# B&R Automation Studio project TD52 (part 30)

```iecst
	(* W9254 Engine cooling water hydraulic pre-heating failure *)
	xMsg9254.Enable	   :=	(xEngType.Type3 OR xEngType.Type4 OR xEngType.Type6)
					AND		Para.bT_HW_Su_PreH_ECW_Active
					AND	(	(Para.iECW_PreH_Int_Visible = 5)					(* el.+hydr. pre-heating available *)
						 OR (	(Para.iECW_PreH_Int_Visible = 3)				(* only hydr. pre-heating available *)
							 AND NOT (Para.rT_ECW_HydrPreH_LimLo = 0.0)	)	);	(* monitoring deactivated if hydr. pre-heating only and Para.rT_ECW_HydrPreH_LimLo = 0.0 *)
	xMsg9254.Set 	   := 	IN_AG.tPB2MM.bParaSetupOk
					AND		bECW_HydrPreH_Dem
					AND (	((IN_AG.tT_ECW.Ai < rT_ECW_HydrPreH_LimLo) AND xSR_PreH_HeatUpDone.Q1)
						 OR	((IN_AG.tT_HW_Su_PreH_ECW.Ai < MM2VIS.rT_HW_Su_PreH_ECW_LimLo) AND IN_AG.tT_HW_Su_PreH_ECW.GoodQual)
						 OR	((IN_AG.tT_HW_Su_PreH_ECW.Ai > MM2VIS.rT_HW_Su_PreH_ECW_LimHi) AND IN_AG.tT_HW_Su_PreH_ECW.GoodQual)	);
	xMsg9254.PT	       := T#0s;
	xMsg9254.Prio 	   := 4;
	xMsg9254.RiskClass := 4;
	xMsg9254.Reset 	   := FALSE;
	xMsg9254();
	MM2VIS.bMsg9254    := xMsg9254.Q;

	(* W9255 Failure high temperature circuit pump 2 (redundant heating water pump) *)
	xMsg9255.Enable	   := Para.bRedHWP_Active;
	xMsg9255.Set 	   := bRedHWP_Fail AND ((iRedHWP_Fail = 2) OR (iRedHWP_Fail = 3));
	xMsg9255.PT	       := T#0s;
	xMsg9255.Prio 	   := 4;
	xMsg9255.RiskClass := 4;
	xMsg9255.Reset	   := FALSE;
	xMsg9255();
	MM2VIS.bMsg9255    := xMsg9255.Q;

	(* W9256 Failure low temperature circuit pump 3 (redundant charge cooler pump) *)
	xMsg9256.Enable	   := Para.bRedCCWP_Active;
	xMsg9256.Set 	   := bRedCCWP_Fail AND ((iRedCCWP_Fail = 2) OR (iRedCCWP_Fail = 3));
	xMsg9256.PT	       := T#0s;
	xMsg9256.Prio 	   := 4;
	xMsg9256.RiskClass := 4;
	xMsg9256.Reset	   := FALSE;
	xMsg9256();
	MM2VIS.bMsg9256    := xMsg9256.Q;

	(* W9257 Failure low temperature circuit pump 4 (redundant charge cooler 2 pump) *)
	xMsg9257.Enable	   := Para.bRedCC2WP_Active;
	xMsg9257.Set 	   := bRedCC2WP_Fail AND ((iRedCC2WP_Fail = 2) OR (iRedCC2WP_Fail = 3));
	xMsg9257.PT	       := T#0s;
	xMsg9257.Prio 	   := 4;
	xMsg9257.RiskClass := 4;
	xMsg9257.Reset	   := FALSE;
	xMsg9257();
	MM2VIS.bMsg9257    := xMsg9257.Q;

	(* W9258 Failure emergency cooling circuit pump 2 (redundant emergency cooler pump) *)
	xMsg9258.Enable	   := Para.bRedEmCWP_Active;
	xMsg9258.Set 	   := bRedEmCWP_Fail AND ((iRedEmCWP_Fail = 2) OR (iRedEmCWP_Fail = 3));
	xMsg9258.PT	       := T#0s;
	xMsg9258.Prio 	   := 4;
	xMsg9258.RiskClass := 4;
	xMsg9258.Reset	   := FALSE;
	xMsg9258();
	MM2VIS.bMsg9258    := xMsg9258.Q;

	(* W9279 Failure emergency cooling circuit pump 1 (emergency cooler pump) *)
	xTOF_EmCWP_Fail(IN:= IN_AG.tEmCWP_Op.Di OR bNoMon4BlackStart, PT:= T#10s);			(*pump operation feedback has to disappear for 10s to trigger warning, ignore feedback in case of black start*)
	xTON_EmCWP_Dem(IN:= IN_AG.bEmCWP_Dem, PT:= T#175s);
	HBT_8 := xTOF_EmCWP_Fail.Q OR (IN_AG.bEng_Aux_Dem AND IN_AG.bEmCWP_Dem AND HBT_8);	(*case 1: HBT_8 -> monitoring activated as soon as pump operation feedback is active for the first time*)

	xMsg9279.Enable	   := TRUE;
	IF NOT Para.bRedEmCWP_Active THEN
		xMsg9279.Set   := (xTON_EmCWP_Dem.Q OR HBT_8) AND NOT xTOF_EmCWP_Fail.Q AND IN_AG.bEmCWP_Dem;		(*case 2: xTON_EmCWP_Dem -> monitoring activated with delay after pump demand*)
	ELSE
		xMsg9279.Set   := bRedEmCWP_Fail AND ((iRedEmCWP_Fail = 1) OR (iRedEmCWP_Fail = 3));
	END_IF;
	xMsg9279.PT	       := T#2s;
	xMsg9279.Prio 	   := 4;
	xMsg9279.RiskClass := 4;
	xMsg9279.Reset	   := FALSE;
	xMsg9279();
	MM2VIS.bMsg9279    := xMsg9279.Q;

	(* W9280 Maximum number of failed post coolings for turbocharger exceeded; inspection of turbocharger required *)
	xMsg9280.Enable	   := FALSE AND IN_AG.tPB2MM.bParaSetupOk;
	xMsg9280.Set 	   := iCnt_TC_rel_A >= Para.iCnt_TC_Inspection_Hi;			(* if only one TC, counter for bank A is used *)
	xMsg9280.PT	       := T#0s;
	xMsg9280.Prio 	   := 4;
	xMsg9280.RiskClass := 4;
	xMsg9280.Reset	   := FALSE;
	xMsg9280();
	MM2VIS.bMsg9280    := xMsg9280.Q;

	(* W9281 Maximum number of failed post coolings for turbocharger at bank A exceeded; inspection of turbocharger required *)
	xMsg9281.Enable	   := xEngType.Type9 AND IN_AG.tPB2MM.bParaSetupOk;
	xMsg9281.Set 	   := iCnt_TC_rel_A >= Para.iCnt_TC_Inspection_Hi;
	xMsg9281.PT	       := T#0s;
	xMsg9281.Prio 	   := 4;
	xMsg9281.RiskClass := 4;
	xMsg9281.Reset	   := FALSE;
	xMsg9281();
	MM2VIS.bMsg9281    := xMsg9281.Q;

	(* W9282 Maximum number of failed post coolings for turbocharger at bank B exceeded; inspection of turbocharger required *)
	xMsg9282.Enable	   := xEngType.Type9 AND IN_AG.tPB2MM.bParaSetupOk;
	xMsg9282.Set 	   := iCnt_TC_rel_B >= Para.iCnt_TC_Inspection_Hi;
	xMsg9282.PT	       := T#0s;
	xMsg9282.Prio 	   := 4;
	xMsg9282.RiskClass := 4;
	xMsg9282.Reset	   := FALSE;
	xMsg9282();
	MM2VIS.bMsg9282    := xMsg9282.Q;

	(* W9283 Failed post cooling for turbocharger detected *)
	xMsg9283.Enable	   := NOT xEngType.Type2 AND IN_AG.tPB2MM.bParaSetupOk;
	xMsg9283.Set 	   := (EDGEPOS(IN_AG.tPB2MM.bSys_Run) AND iSt_TC_PwrInterrupt.0) OR EDGENEG(bTC_CoolDownInterrupt);
	xMsg9283.PT	       := T#0s;
	xMsg9283.Prio 	   := 4;
	xMsg9283.RiskClass := 4;
	xMsg9283.Reset	   := FALSE;
	xMsg9283();
	MM2VIS.bMsg9283    := xMsg9283.Q;

	(* W9303 Measuring signal failure air starter engagement pressure *)
	xMsg9303.Enable	   := xEngType.Type9;
	xMsg9303.Set 	   := bAMM_Pr_AirST_Engage_Ms;
	xMsg9303.PT	       := T#0s;
	xMsg9303.Prio 	   := 4;
	xMsg9303.RiskClass := 4;
	xMsg9303.Reset	   := FALSE;
	xMsg9303();
	MM2VIS.bMsg9303    := xMsg9303.Q;

	(* W9314 Engine cooling water pump circuit breaker tripped *)
	xMsg9314.Enable	   := IN_AG.tPB2MM.bParaSetupOk;
	xMsg9314.Set 	   := NOT IN_AG.tECWP_CB_On.Di;
	xMsg9314.PT	       := T#1s;
	xMsg9314.Prio 	   := 4;
	xMsg9314.RiskClass := 4;
	xMsg9314.Reset	   := FALSE;
	xMsg9314();
	MM2VIS.bMsg9314    := xMsg9314.Q;

	(* W9316 Measuring signal failure cooling water pressure after ECW pump 1 *)
	xMsg9316.Enable	   := Para.bDPr_ECWP_Mon_Active AND IN_AG.tPr_ECWaP1.Exist;
	xMsg9316.Set 	   := NOT IN_AG.tPr_ECWaP1.GoodQual;
	xMsg9316.PT	       := T#1s;
	xMsg9316.Prio 	   := 4;
	xMsg9316.RiskClass := 4;
	xMsg9316.Reset	   := FALSE;
	xMsg9316();
	MM2VIS.bMsg9316    := xMsg9316.Q;

	(* W9317 Measuring signal failure cooling water pressure after ECW pump 2 *)
	xMsg9317.Enable	   := Para.bDPr_ECWP_Mon_Active AND IN_AG.tPr_ECWaP2.Exist;
	xMsg9317.Set 	   := NOT IN_AG.tPr_ECWaP2.GoodQual;
	xMsg9317.PT	       := T#1s;
	xMsg9317.Prio 	   := 4;
	xMsg9317.RiskClass := 4;
	xMsg9317.Reset	   := FALSE;
	xMsg9317();
	MM2VIS.bMsg9317    := xMsg9317.Q;

	(* W9322 Fresh oil tank level low (2nd level switch) *)
	xMsg9322.Enable	   := IN_AG.tL_FreshOilTank_LoLo.GoodQual;
	xMsg9322.Set 	   := NOT IN_AG.tL_FreshOilTank_LoLo.Di;
	xMsg9322.PT	       := T#0s;
	xMsg9322.Prio 	   := 4;
	xMsg9322.RiskClass := 4;
	xMsg9322.Reset	   := FALSE;
	xMsg9322();
	MM2VIS.bMsg9322    := xMsg9322.Q;

	(* W9323 Fresh oil day tank level low *)
	xMsg9323.Enable	   := IN_AG.tPB2MM.bParaSetupOk;
	xMsg9323.Set 	   := (IN_AG.tL_DayOilTank_Lo.GoodQual AND NOT IN_AG.tL_DayOilTank_Lo.Di)
					   OR (IN_AG.tL_DayOilTank.GoodQual AND (MM2VIS.rV_DayOilTank < Para.rV_DayOilTank_LimLo) AND (Para.rV_DayOilTank_LimLo > 0)) ;		(*New at V4.12*)
	xMsg9323.PT	       := T#0s;
	xMsg9323.Prio 	   := 4;
	xMsg9323.RiskClass := 4;
	xMsg9323.Reset	   := FALSE;
	xMsg9323();
	MM2VIS.bMsg9323    := xMsg9323.Q;

	(* W9324 Fresh oil day tank level low (2nd level switch) *)
	xMsg9324.Enable	   := IN_AG.tL_DayOilTank_LoLo.GoodQual;
	xMsg9324.Set 	   := NOT IN_AG.tL_DayOilTank_LoLo.Di;
	xMsg9324.PT	       := T#0s;
	xMsg9324.Prio 	   := 4;
	xMsg9324.RiskClass := 4;
	xMsg9324.Reset	   := FALSE;
	xMsg9324();
	MM2VIS.bMsg9324    := xMsg9324.Q;

	(* W9325 Overfill prevention device fresh oil day tank tripped *)
	xMsg9325.Enable	   := IN_AG.tOF_DayOilTank.GoodQual;
	xMsg9325.Set 	   := NOT IN_AG.tOF_DayOilTank.Di;
	xMsg9325.PT	       := T#0s;
	xMsg9325.Prio 	   := 4;
	xMsg9325.RiskClass := 4;
	xMsg9325.Reset	   := FALSE;
	xMsg9325();
	MM2VIS.bMsg9325    := xMsg9325.Q;

	(* W9326 Waste oil day tank level high *)
	xMsg9326.Enable	   := IN_AG.tL_WasteOilDayTank_Hi.GoodQual;
	xMsg9326.Set 	   := NOT IN_AG.tL_WasteOilDayTank_Hi.Di;
	xMsg9326.PT	       := T#0s;
	xMsg9326.Prio 	   := 4;
	xMsg9326.RiskClass := 4;
	xMsg9326.Reset	   := FALSE;
	xMsg9326();
	MM2VIS.bMsg9326    := xMsg9326.Q;

	(* W9327 Overfill prevention device waste oil day tank tripped *)
	xMsg9327.Enable	   := IN_AG.tOF_WasteOilDayTank.GoodQual;
	xMsg9327.Set 	   := NOT IN_AG.tOF_WasteOilDayTank.Di;
	xMsg9327.PT	       := T#0s;
	xMsg9327.Prio 	   := 4;
	xMsg9327.RiskClass := 4;
	xMsg9327.Reset	   := FALSE;
	xMsg9327();
	MM2VIS.bMsg9327    := xMsg9327.Q;

	(* W9328 Fresh oil pump oil pressure maximum *)
	xMsg9328.Enable	   := IN_AG.tPS_FreshOilPump_Hi.GoodQual;
	xMsg9328.Set 	   := NOT IN_AG.tPS_FreshOilPump_Hi.Di;
	xMsg9328.PT	       := T#0s;
	xMsg9328.Prio 	   := 4;
	xMsg9328.RiskClass := 4;
	xMsg9328.Reset	   := FALSE;
	xMsg9328();
	MM2VIS.bMsg9328    := xMsg9328.Q;

	(* W9332 Take oil sample *)
	xMsg9332.Enable	   := Para.bEO_Management_Active AND IN_AG.tPB2MM.bParaSetupOk;
	xMsg9332.Set 	   := bMsg9332_set;
	xMsg9332.PT	       := T#0s;
	xMsg9332.Prio 	   := 4;
	xMsg9332.RiskClass := 4;
	xMsg9332.Reset	   := TRUE;
	xMsg9332();
	MM2VIS.bMsg9332    := xMsg9332.Q;

	(* W9333 Take coolant sample *)
	xMsg9333.Enable	   := Para.bCW_Management_Active AND IN_AG.tPB2MM.bParaSetupOk;
	xMsg9333.Set 	   := bMsg9333_set;
	xMsg9333.PT	       := T#0s;
	xMsg9333.Prio 	   := 4;
	xMsg9333.RiskClass := 4;
	xMsg9333.Reset	   := TRUE;
	xMsg9333();
	MM2VIS.bMsg9333    := xMsg9333.Q;

	(* W9334 Buffer battery 1 voltage low *)
	xMsg9334.Enable	   := IN_AG.tPB2MM.bParaSetupOk AND ((Para.iBatMon_Mode = 1) OR (Para.iBatMon_Mode = 2));
	xMsg9334.Set 	   := bAMM_U_BufferBat1_Lo;
	xMsg9334.PT	       := T#0s;
	xMsg9334.Prio 	   := 4;
	xMsg9334.RiskClass := 4;
	xMsg9334.Reset	   := FALSE;
	xMsg9334();
	MM2VIS.bMsg9334    := xMsg9334.Q;

	(* W9335 Buffer battery 2 voltage low *)
	xMsg9335.Enable	   := IN_AG.tPB2MM.bParaSetupOk AND (Para.iBatMon_Mode = 2);
	xMsg9335.Set 	   := bAMM_U_BufferBat2_Lo;
	xMsg9335.PT	       := T#0s;
	xMsg9335.Prio 	   := 4;
	xMsg9335.RiskClass := 4;
	xMsg9335.Reset	   := FALSE;
	xMsg9335();
	MM2VIS.bMsg9335    := xMsg9335.Q;

	(* W9336 Battery charging device malfunction *)
	xMsg9336.Enable	   := IN_AG.tPB2MM.bParaSetupOk;
	xMsg9336.Set 	   := NOT IN_AG.tBatChargeDev_Ok.Di;
	xMsg9336.PT	       := T#10s;
	xMsg9336.Prio 	   := 4;
	xMsg9336.RiskClass := 4;
	xMsg9336.Reset	   := FALSE;
	xMsg9336();
	MM2VIS.bMsg9336    := xMsg9336.Q;

	(* W9352 Oil quality sensor - Measurement signal failure, return to regular sampling interval *)
	xMsg9352.Enable	   := (Para.iOQS_Config = 1) AND IN_AG.tPB2MM.bParaSetupOk AND NOT IN_AG.bSimWinMOD_Active;
	xMsg9352.Set 	   := bAMM_OQS_OC_MSF;
	xMsg9352.PT	       := T#0s;
	xMsg9352.Prio 	   := 4;
	xMsg9352.RiskClass := 4;
	xMsg9352.Reset	   := FALSE;
	xMsg9352();
	MM2VIS.bMsg9352    := xMsg9352.Q;

	(* W9353 Oil quality sensor - Oil quality warning, return to regular sampling interval *)
	xMsg9353.Enable	   := (Para.iOQS_Config = 1) AND IN_AG.tPB2MM.bParaSetupOk AND NOT IN_AG.bSimWinMOD_Active;
	xMsg9353.Set 	   := bAMM_OQS_OC_ValueLo;
	xMsg9353.PT	       := T#0s;
	xMsg9353.Prio 	   := 4;
	xMsg9353.RiskClass := 4;
	xMsg9353.Reset	   := FALSE;
	xMsg9353();
	MM2VIS.bMsg9353    := xMsg9353.Q;

	(* W9354 Oil quality sensor  Critical oil quality warning, return to regular sampling interval *)
	xMsg9354.Enable	   := (Para.iOQS_Config = 1) AND IN_AG.tPB2MM.bParaSetupOk AND NOT IN_AG.bSimWinMOD_Active;
	xMsg9354.Set 	   := bAMM_OQS_OC_ValueLo1;
	xMsg9354.PT	       := T#0s;
	xMsg9354.Prio 	   := 4;
	xMsg9354.RiskClass := 4;
	xMsg9354.Reset	   := FALSE;
	xMsg9354();
	MM2VIS.bMsg9354    := xMsg9354.Q;

	(* W9355 Oil quality sensor  Increased oil aging, return to regular sampling interval *)
	xMsg9355.Enable	   := (Para.iOQS_Config = 1) AND IN_AG.tPB2MM.bParaSetupOk AND NOT IN_AG.bSimWinMOD_Active;
	xMsg9355.Set 	   := bAMM_OQS_OC_TendencyHi;
	xMsg9355.PT	       := T#0s;
	xMsg9355.Prio 	   := 4;
	xMsg9355.RiskClass := 4;
	xMsg9355.Reset	   := FALSE;
	xMsg9355();
	MM2VIS.bMsg9355    := xMsg9355.Q;

	(* W9356 Oil quality sensor - Critical oil aging, return to regular sampling interval *)
	xMsg9356.Enable	   := (Para.iOQS_Config = 1) AND IN_AG.tPB2MM.bParaSetupOk AND NOT IN_AG.bSimWinMOD_Active;
	xMsg9356.Set 	   := bAMM_OQS_OC_TendencyHi1;
	xMsg9356.PT	       := T#0s;
	xMsg9356.Prio 	   := 4;
	xMsg9356.RiskClass := 4;
	xMsg9356.Reset	   := FALSE;
	xMsg9356();
	MM2VIS.bMsg9356    := xMsg9356.Q;

	(* W9357 Control battery voltage low *)
	xMsg9357.Enable	   := IN_AG.tPB2MM.bParaSetupOk AND (iNr_CtrlBat_Used > 0);
	xMsg9357.Set 	   := bAMM_U_CtrlBat_Lo_Coll;
	xMsg9357.PT	       := T#0s;
	xMsg9357.Prio 	   := 4;
	xMsg9357.RiskClass := 4;
	xMsg9357.Reset	   := FALSE;
	xMsg9357();
	MM2VIS.bMsg9357    := xMsg9357.Q;

	(* W9358 Control battery charging device malfunction *)
	bAMM_CtrlBat_ChargeDev_Fail		:=	FALSE;
	FOR iIdx_CtrlBat := 1 TO iNum_CtrlBatMon DO
		bAMM_CtrlBat_ChargeDev_Fail	:=	NOT IN_AG.tCtrlBat_ChargeDev_Ok[iIdx_CtrlBat].Di OR bAMM_CtrlBat_ChargeDev_Fail;
		IF NOT IN_AG.tCtrlBat_ChargeDev_Ok[iIdx_CtrlBat].Di THEN
			MM2VIS.sCtrlBat_ChargeDev_LocFault	:=	IN_AG.sLocIdent_CtrlBatMon[iIdx_CtrlBat];
		END_IF;
	END_FOR;
	xMsg9358.Enable	   := IN_AG.tPB2MM.bParaSetupOk AND (iNr_CtrlBat_Used > 0);
	xMsg9358.Set 	   := bAMM_CtrlBat_ChargeDev_Fail;
	xMsg9358.PT	       := T#10s;
	xMsg9358.Prio 	   := 4;
	xMsg9358.RiskClass := 4;
	xMsg9358.Reset	   := FALSE;
	xMsg9358();
	MM2VIS.bMsg9358    := xMsg9358.Q;

	(* W9359 Oil pressure before centrifuge (oil filter unit) minimum *)
	xMsg9359.Enable	   := Para.bOilFiltUnit_Exist AND Para.bPr_OFUbCentrifuge_Active;
	xMsg9359.Set 	   := bAMM_Pr_OFUbCentrifuge_Lo;
	xMsg9359.PT	       := T#2s;
	xMsg9359.Prio 	   := 4;
	xMsg9359.RiskClass := 4;
	xMsg9359.Reset	   := FALSE;
	xMsg9359();
	MM2VIS.bMsg9359    := xMsg9359.Q;

	(*W9362 Fresh Oil Tank Signal Failure V4.12 *)
	xMsg9362.Enable		:=  Para.bOilTankMonitoring AND Para.rFreshOilTank_Type > 0;
	xMsg9362.Set 	   := NOT IN_AG.tL_FreshOilTank.GoodQual;
	xMsg9362.PT	       := T#2s;
	xMsg9362.Prio 	   := 4;
	xMsg9362.RiskClass := 4;
	xMsg9362.Reset	   := FALSE;
	xMsg9362();
	MM2VIS.bMsg9362    := xMsg9362.Q;

	(*W9363 Waste Oil Tank Signal Failure V4.12 *)
	xMsg9363.Enable		:=  Para.bOilTankMonitoring AND Para.rWasteOilTank_Type > 0;
	xMsg9363.Set 	   := NOT IN_AG.tL_WasteOilTank.GoodQual;
	xMsg9363.PT	       := T#2s;
	xMsg9363.Prio 	   := 4;
	xMsg9363.RiskClass := 4;
	xMsg9363.Reset	   := FALSE;
	xMsg9363();
	MM2VIS.bMsg9363    := xMsg9363.Q;

	(*W9364 Fresh Oil Tank Signal Failure V4.12 *)
	xMsg9364.Enable		:=  Para.bOilTankMonitoring AND Para.rDayOilTank_Type > 0;
	xMsg9364.Set 	   := NOT IN_AG.tL_DayOilTank.GoodQual;
	xMsg9364.PT	       := T#2s;
	xMsg9364.Prio 	   := 4;
	xMsg9364.RiskClass := 4;
	xMsg9364.Reset	   := FALSE;
	xMsg9364();
	MM2VIS.bMsg9364    := xMsg9364.Q;

	(*W9369 Failure auxiliaries supply voltage engine V4.12 *)
	xMsg9369.Enable		:= IN_AG.tPB2MM.bParaSetupOk;
	xMsg9369.Set		:= (NOT IN_AG.tAuxV_Eng_ok.Di) AND IN_AG.tAuxV_Eng_ok.GoodQual AND IN_AG.tMnsOk.Di AND IN_AG.tMnsOk.GoodQual;
	xMsg9369.PT			:= T#1m;
	xMsg9369.Prio		:= 4;
	xMsg9369.RiskClass	:= 4;
	xMsg9369.Reset		:= FALSE;
	xMsg9369();
	MM2VIS.bMsg9369    := xMsg9369.Q;

	(*W9378 Oil refill volume maximum *)
	xMsg9378.Enable		:= IN_AG.tPB2MM.bParaSetupOk;
	xMsg9378.Set		:= bAMM_Vol_OilRefill_Hi;
	xMsg9378.PT			:= T#0s;
	xMsg9378.Prio		:= 4;
	xMsg9378.RiskClass	:= 4;
	xMsg9378.Reset		:= FALSE;
	xMsg9378();
	MM2VIS.bMsg9378    	:= xMsg9378.Q;

	(*W9390 Oil temperature before engine start too low *)
	xMsg9390.Enable		:= IN_AG.tPB2MM.bParaSetupOk;
	xMsg9390.Set		:= bAMM_T_EO_PreH_EngStart_Lo;
	xMsg9390.PT			:= T#0s;
	xMsg9390.Prio		:= 4;
	xMsg9390.RiskClass	:= 4;
	xMsg9390.Reset		:= NOT bAMM_T_EO_PreH_EngStart_Lo;
	xMsg9390();
	MM2VIS.bMsg9390    	:= xMsg9390.Q;

	(* A9435 Fire detection system - System failure *)
	xMsg9435.Enable	   	:= IN_AG.tPB2MM.bParaSetupOk AND IN_AG.bSafetyPLC_Active;			(* SAFETY PLC *)
	xMsg9435.Set	  	:= NOT IN_AG.tFireSysErr.Di;
	xMsg9435.PT	       	:= T#240s;
	xMsg9435.Prio	   	:= 3;
	xMsg9435.RiskClass	:= 4;
	xMsg9435.Reset	   	:= FALSE;
	xMsg9435();
	MM2VIS.bMsg9435		:= xMsg9435.Q;

	(* A9436 Gas detection system - System failure *)
	xMsg9436.Enable	   	:= IN_AG.tPB2MM.bParaSetupOk AND IN_AG.bSafetyPLC_Active;			(* SAFETY PLC *)
	xMsg9436.Set	  	:= NOT IN_AG.tGasSysErr.Di;
	xMsg9436.PT	       	:= T#240s;
	xMsg9436.Prio	   	:= 3;
	xMsg9436.RiskClass	:= 4;
	xMsg9436.Reset	   	:= FALSE;
	xMsg9436();
	MM2VIS.bMsg9436		:= xMsg9436.Q;

	(* W9560 Fire detection system - System failure *)
	xMsg9560.Enable	   	:= IN_AG.tPB2MM.bParaSetupOk AND IN_AG.bSafetyPLC_Active;			(* SAFETY PLC *)
	xMsg9560.Set	  	:= NOT IN_AG.tFireSysErr.Di;
	xMsg9560.PT	       	:= T#0s;
	xMsg9560.Prio	   	:= 4;
	xMsg9560.RiskClass	:= 4;
	xMsg9560.Reset	   	:= FALSE;
	xMsg9560();
	MM2VIS.bMsg9560		:= xMsg9560.Q;

	(* W9561 Gas detection system - System failure *)
	xMsg9561.Enable	   	:= IN_AG.tPB2MM.bParaSetupOk AND IN_AG.bSafetyPLC_Active;			(* SAFETY PLC *)
	xMsg9561.Set	  	:= NOT IN_AG.tGasSysErr.Di;
	xMsg9561.PT	       	:= T#0s;
	xMsg9561.Prio	   	:= 4;
	xMsg9561.RiskClass	:= 4;
	xMsg9561.Reset	   	:= FALSE;
	xMsg9561();
	MM2VIS.bMsg9561		:= xMsg9561.Q;

	(*---------------------------------------------------------------------------*)
	(* operating messages > AMM *)

	(* B1249 starter engine on *)
	xMsg1249.Enable		:=	TRUE;
	xMsg1249.Set		:= 	(OUT_AG.bEng_Start AND xEngType.Type9) OR (OUT_AG.tEleStarter_Dem.Do AND NOT xEngType.Type9);
	xMsg1249.Reset		:=	TRUE;
	xMsg1249();
	MM2VIS.bMsg1249		:=	xMsg1249.Q;

	(* B1250 starter engine off *)
	xMsg1250.Enable		:=	IN_AG.tPB2MM.bSys_Run;
	xMsg1250.Set		:=	NOT MM2VIS.bMsg1249;
	xMsg1250.Reset		:=	TRUE;
	xMsg1250();
	MM2VIS.bMsg1250		:= xMsg1250.Q;

	(* B1257 demand engine cooling water pump on *)
	xMsg1257.Enable		:=	TRUE;
	xMsg1257.Set		:=	    OUT_AG.tECWP1Dem.Do;
	xMsg1257.Reset		:=	TRUE;
	xMsg1257();
	MM2VIS.bMsg1257		:= xMsg1257.Q;

	(* B1258 demand engine cooling water pump off *)
	xMsg1258.Enable		:=	IN_AG.tPB2MM.bSys_Run;
	xMsg1258.Set		:=	NOT OUT_AG.tECWP1Dem.Do;
	xMsg1258.Reset		:=	TRUE;
	xMsg1258();
	MM2VIS.bMsg1258		:= xMsg1258.Q;

	(* B1259 demand oil pump on *)
	xMsg1259.Enable		:=	TRUE;
	xMsg1259.Set		:=	OUT_AG.tEOP1AC_Dem.Do;
	xMsg1259.Reset		:=	TRUE;
	xMsg1259();
	MM2VIS.bMsg1259		:= xMsg1259.Q;

	(* B1260 demand oil pump off *)
	xMsg1260.Enable		:=	IN_AG.tPB2MM.bSys_Run;
	xMsg1260.Set		:=	NOT OUT_AG.tEOP1AC_Dem.Do;
	xMsg1260.Reset		:=	TRUE;
	xMsg1260();
	MM2VIS.bMsg1260		:= xMsg1260.Q;

	(* B1261 demand oil pump (DC) on *)
	xMsg1261.Enable		:=	NOT xEngType.Type9;
	xMsg1261.Set		:=	    OUT_AG.tEOP1DC_Dem.Do;
	xMsg1261.Reset		:=	TRUE;
	xMsg1261();
	MM2VIS.bMsg1261		:= xMsg1261.Q;

	(* B1262 demand oil pump (DC) off *)
	xMsg1262.Enable		:=	IN_AG.tPB2MM.bSys_Run AND NOT xEngType.Type9;
	xMsg1262.Set		:=	NOT OUT_AG.tEOP1DC_Dem.Do;
	xMsg1262.Reset		:=	TRUE;
	xMsg1262();
	MM2VIS.bMsg1262		:= xMsg1262.Q;

	(* B1263 demand turbo charger oil pump on *)
	xMsg1263.Enable		:=	TRUE;
	xMsg1263.Set		:=  OUT_AG.tTC_EOP_On.Do OR OUT_AG.tTC_EOP_OnUSV.Do;
	xMsg1263.Reset		:=	TRUE;
	xMsg1263();
	MM2VIS.bMsg1263		:= xMsg1263.Q;

	(* B1264 demand turbo charger oil pump off *)
	xMsg1264.Enable		:=	IN_AG.tPB2MM.bSys_Run AND xEngType.Type9;
	xMsg1264.Set		:=	NOT OUT_AG.tTC_EOP_On.Do AND NOT OUT_AG.tTC_EOP_OnUSV.Do;
	xMsg1264.Reset		:=	TRUE;
	xMsg1264();
	MM2VIS.bMsg1264		:= xMsg1264.Q;

	(* B1281 demand engine cooling water preheating pump on *)
	xMsg1281.Enable		:=	TRUE;
	xMsg1281.Set		:=	    OUT_AG.tECWP_PreH_Dem.Do;
	xMsg1281.Reset		:=	TRUE;
	xMsg1281();
	MM2VIS.bMsg1281		:= xMsg1281.Q;

	(* B1282 demand engine cooling water preheating pump off *)
	xMsg1282.Enable		:=	IN_AG.tPB2MM.bSys_Run;
	xMsg1282.Set		:=	NOT OUT_AG.tECWP_PreH_Dem.Do;
	xMsg1282.Reset		:=	TRUE;
	xMsg1282();
	MM2VIS.bMsg1282		:= xMsg1282.Q;

	(* B1292 Manual operating auxiliaries control (Handbedienebene) active *)
	xMsg1292.Enable		:=	IN_AG.tPB2MM.bSys_Run;
	xMsg1292.Set		:=	bMsg1292_Set;
	xMsg1292.Reset		:=	TRUE;
	xMsg1292();
	MM2VIS.bMsg1292		:= xMsg1292.Q;

	(* B2809 preheating valve opened *)
	xMsg2809.Enable		:=	IN_AG.tPB2MM.bSys_Run;
	xMsg2809.Set		:=	IN_AG.tECW_PreHV_Opened.Di;
	xMsg2809.Reset		:=	TRUE;
	xMsg2809();
	MM2VIS.bMsg2809		:= xMsg2809.Q;

	(* B2810 Preheating valve closed *)
	xMsg2810.Enable		:=	bECW_PreHV_Active;
	xMsg2810.Set		:=	IN_AG.tECW_PreHV_Closed.Di;
	xMsg2810.Reset		:=	TRUE;
	xMsg2810();
	MM2VIS.bMsg2810		:= xMsg2810.Q;

	(* B2931 Active Cooling Program in operation *)
	xMsg2931.Enable		:=	Para.bACP_Enable;
	xMsg2931.Set		:=	bACP_Start AND NOT bACP_Cmp;
	xMsg2931.Reset		:=	TRUE;
	xMsg2931();
	MM2VIS.bMsg2931		:= xMsg2931.Q;

	(* B2932 Active Cooling Program finished *)
	xMsg2932.Enable		:=	Para.bACP_Enable;
	xMsg2932.Set		:=	bACP_Cmp;
	xMsg2932.Reset		:=	TRUE;
	xMsg2932();
	MM2VIS.bMsg2932		:= xMsg2932.Q;

	(* B2933 Active Cooling Program cancelled *)
	xF_TRIG_ACP_Start(CLK := bACP_Start);
	xMsg2933.Enable		:=	Para.bACP_Enable;
	xMsg2933.Set		:=	xF_TRIG_ACP_Start.Q AND NOT bACP_Cmp;
	xMsg2933.Reset		:=	TRUE;
	xMsg2933();
	MM2VIS.bMsg2933		:= xMsg2933.Q;

	(* B2956 Demand engine oil preheating valve open *)
	xMsg2956.Enable		:=	IN_AG.tPB2MM.bSys_Run
						AND xEngType.Type9;
	xMsg2956.Set		:=	OUT_AG.tEOF_PreheatRel.Do;
	xMsg2956.Reset		:=	TRUE;
	xMsg2956();
	MM2VIS.bMsg2956		:= xMsg2956.Q;

	(* B2957 Demand engine oil preheating valve close *)
	xMsg2957.Enable		:=	IN_AG.tPB2MM.bSys_Run
						AND xEngType.Type9;
	xMsg2957.Set		:=	NOT OUT_AG.tEOF_PreheatRel.Do;
	xMsg2957.Reset		:=	TRUE;
	xMsg2957();
	MM2VIS.bMsg2957		:= xMsg2957.Q;

	(* B2978 Blow-by blower on *)
	xMsg2978.Enable		:=	xEngType.Type9;
	xMsg2978.Set		:=	OUT_AG.tBbBlower.Do;
	xMsg2978.Reset		:=	TRUE;
	xMsg2978();
	MM2VIS.bMsg2978		:= xMsg2978.Q;

	(* B2979 Blow-by blower off *)
	xMsg2979.Enable		:=	xEngType.Type9;
	xMsg2979.Set		:=	NOT OUT_AG.tBbBlower.Do;
	xMsg2979.Reset		:=	TRUE;
	xMsg2979();
	MM2VIS.bMsg2979		:= xMsg2979.Q;

	(* B3300 blocking acknowledgement by starter temperature *)
	xMsg3300.Enable		:=	TRUE;
	xMsg3300.Set		:=	OUT_AG.bLockAckStarter;
	xMsg3300.Reset		:=	TRUE;
	xMsg3300();
	MM2VIS.bMsg3300		:= xMsg3300.Q;

	(* B9001 Oil sample taken *)
	xMsg9001.Enable		:=	Para.bEO_Management_Active AND IN_AG.tPB2MM.bParaSetupOk;
	xMsg9001.Set		:=	bMsg9001_set;
	xMsg9001.Reset		:=	TRUE;
	xMsg9001();
	MM2VIS.bMsg9001		:= xMsg9001.Q;

	(* B9002 Oil exchanged *)
	xMsg9002.Enable		:=	Para.bEO_Management_Active AND IN_AG.tPB2MM.bParaSetupOk;
	xMsg9002.Set		:=	bMsg9002_set;
	xMsg9002.Reset		:=	TRUE;
	xMsg9002();
	MM2VIS.bMsg9002		:= xMsg9002.Q;

	(* B9003 Coolant sample taken *)
	xMsg9003.Enable		:=	Para.bCW_Management_Active AND IN_AG.tPB2MM.bParaSetupOk;
	xMsg9003.Set		:=	bMsg9003_set;
	xMsg9003.Reset		:=	TRUE;
	xMsg9003();
	MM2VIS.bMsg9003		:= xMsg9003.Q;

	(* B9048 Coolant exchanged *)
	xMsg9048.Enable		:=	Para.bCW_Management_Active AND IN_AG.tPB2MM.bParaSetupOk;
	xMsg9048.Set		:=	bMsg9048_set;
	xMsg9048.Reset		:=	TRUE;
	xMsg9048();
	MM2VIS.bMsg9048		:= xMsg9048.Q;

	(* B9067 Oil sampling interval extended *)
	xMsg9067.Enable		:=	(Para.iOQS_Config = 1) AND IN_AG.tPB2MM.bParaSetupOk AND NOT IN_AG.bSimWinMOD_Active;
	xMsg9067.Set		:=	bOpMsg_ExtendOilSampleOh;
	xMsg9067.Reset		:=	TRUE;
	xMsg9067();
	MM2VIS.bMsg9067		:= xMsg9067.Q;

	(* B9069 Buffer battery test in progress *)
	xMsg9069.Enable		:= IN_AG.tPB2MM.bParaSetupOk AND (Para.iBatMon_Mode > 0);
	xMsg9069.Set		:= MM2VIS.bBatMon_TestRunning;
	xMsg9069.Reset		:= TRUE;
	xMsg9069();
	MM2VIS.bMsg9069		:= xMsg9069.Q;

	(* B9070 Control battery test in progress *)
	xMsg9070.Enable		:= IN_AG.tPB2MM.bParaSetupOk AND (iNr_CtrlBat_Used > 0);
	xMsg9070.Set		:= MM2VIS.bCtrlBatMon_TestRunning;
	xMsg9070.Reset		:= TRUE;
	xMsg9070();
	MM2VIS.bMsg9070		:= xMsg9070.Q;

	(* B9074 Tooth to tooth position *)
	xMsg9074.Enable		:= IN_AG.tPB2MM.bParaSetupOk;
	xMsg9074.Set		:= FALSE; // warning message for tooth to tooth detection. Not used yet, already set up in the HMI
	xMsg9074.Reset		:= TRUE;
	xMsg9074();
	MM2VIS.bMsg9074		:= xMsg9074.Q;

	(* B9088 Purge cranking cycle successful *)
	xMsg9088.Enable		:= IN_AG.tPB2MM.bParaSetupOk;
	xMsg9088.Set		:= (bStartScavSflMsg AND xEngType.Type3) OR (bMsg9088_T6_set AND xEngType.Type6);
	xMsg9088.Reset		:= TRUE;
	xMsg9088();
	MM2VIS.bMsg9088 	:= xMsg9088.Q;

	(* B9089 Starter motor 1 did not engage *)
	xMsg9089.Enable		:= IN_AG.tPB2MM.bParaSetupOk AND Para.rU_StarterMon_LimLo <> 0.0;
	xMsg9089.Set		:= bEleStarterFail_Num[1];
	xMsg9089.Reset		:= TRUE;
	xMsg9089();
	MM2VIS.bMsg9089		:= xMsg9089.Q;

	(* B9090 Starter motor 2 did not engage *)
	xMsg9090.Enable		:= IN_AG.tPB2MM.bParaSetupOk AND Para.rU_StarterMon_LimLo <> 0.0;
	xMsg9090.Set		:= bEleStarterFail_Num[2];
	xMsg9090.Reset		:= TRUE;
	xMsg9090();
	MM2VIS.bMsg9090		:= xMsg9090.Q;

	(* B9091 Starter motor 3 did not engage *)
	xMsg9091.Enable		:= IN_AG.tPB2MM.bParaSetupOk AND Para.rU_StarterMon_LimLo <> 0.0;
	xMsg9091.Set		:= bEleStarterFail_Num[3];
	xMsg9091.Reset		:= TRUE;
	xMsg9091();
	MM2VIS.bMsg9091		:= xMsg9091.Q;

	(* B9096 Starter overheated *)
	xMsg9096.Enable		:= IN_AG.tPB2MM.bParaSetupOk AND xEngType.Type6;
	xMsg9096.Set		:= bMsg9096_set AND bMsg9096_enable;
	xMsg9096.Reset		:= TRUE;
	xMsg9096();
	MM2VIS.bMsg9096		:= xMsg9096.Q;
	MM2VIS.iNum_Msg9096	:= bMsg9096_iTi_ST_UntRelDur;

	(* B9097 Purge cranking cycle initiated *)
	xMsg9097.Enable		:= IN_AG.tPB2MM.bParaSetupOk AND xEngType.Type6;
	xMsg9097.Set		:= bMsg9097_set;
	xMsg9097.Reset		:= TRUE;
	xMsg9097();
	MM2VIS.bMsg9097		:= xMsg9097.Q;

	(*W9513 Failure engine oil refilling *)
	xMsg9513.Enable 	:= IN_AG.tPB2MM.bParaSetupOk ;
	xMsg9513.Set 		:= bAMM_9513;
	xMsg9513.PT 		:= Para.tiEO_Refill_TimeMax;
	xMsg9513.Prio 		:= 4;
	xMsg9513.Reset 		:= FALSE;
	xMsg9513();
	MM2VIS.bMsg9513 	:= xMsg9513.Q;

	(* B template
	xMsg.Enable		:=	TRUE;
	xMsg.Set		:=	bBool;
	xMsg.Reset		:=	TRUE;
	xMsg();
	MM2VIS.bMsg		:=	xMsg.Q;
	*)

	(*---------------------------------------------------------------------------*)
	(* general alarms for further module operations *)
	bGnlTrip1		:= OUT_AG.tAG2AB.bGnlTrip1   OR IN_AG.tAB2AG.bGnlTrip1;
	bGnlTrip2		:= OUT_AG.tAG2AB.bGnlTrip2   OR IN_AG.tAB2AG.bGnlTrip2;
	bGnlTrip3		:= OUT_AG.tAG2AB.bGnlTrip3   OR IN_AG.tAB2AG.bGnlTrip3;
	bGnlWarning		:= OUT_AG.tAG2AB.bGnlWarning OR IN_AG.tAB2AG.bGnlWarning;

	bGnlTrip		:= bGnlTrip1 OR bGnlTrip2 OR bGnlTrip3;

	(*******************************************************************************)

END_PROGRAM
```

#### MsgAGInit.st
```iecst
(*******************************************************************************
Msg_AG	 			 alarms generation auxiliaries general

This code is confidential and proprietary to the INNIO Company.
It may not be used in any form, or reproduced in any manner,
without written permission of the INNIO Company.
Copyright, INNIO Company, 2022

Customized modifications: -
------------------------

History:
-------
V0.00.0	29.07.2011	lettenb.	new
V4.12.0	21.12.2022	Perktold	added W9369 Failure auxiliaries supply voltage engine

Instructions for use:
--------------------
1) declare alarm with function block "Msg"

2) use template to create a new alarm, substitue 0000 by message number:

	xMsg0000.Num		:=	0000;					alarm number
	xMsg0000.AmmSysAdr	:=  iAdrAmmBase2MM;			do not change
	xMsg0000.AmmOutAdr	:=  iAdrMM2AmmBase;			do not change

3) 	set alarm number

Outstandings:
------------
(*******************************************************************************)
PROGRAM _INIT

	bPLC_Startup := FALSE;

	iAdrAmmBase2MM		:=  ADR(IN_AG.tAB2AG);
	iAdrMM2AmmBase		:=  ADR(OUT_AG.tAG2AB);

	(*---------------------------------------------------------------------------*)
	xMsg1017.Num		:=	1017;
	xMsg1017.AmmInAdr	:=  iAdrAmmBase2MM;
	xMsg1017.AmmOutAdr	:=  iAdrMM2AmmBase;

	xMsg1018.Num		:=  1018;
	xMsg1018.AmmInAdr	:=  iAdrAmmBase2MM;
	xMsg1018.AmmOutAdr	:=  iAdrMM2AmmBase;

	xMsg1020.Num		:=  1020;
	xMsg1020.AmmInAdr	:=  iAdrAmmBase2MM;
	xMsg1020.AmmOutAdr	:=  iAdrMM2AmmBase;

	xMsg1023.Num		:=  1023;
	xMsg1023.AmmInAdr	:=  iAdrAmmBase2MM;
	xMsg1023.AmmOutAdr	:=  iAdrMM2AmmBase;

	xMsg1043.Num		:=	1043;
	xMsg1043.AmmInAdr	:=  iAdrAmmBase2MM;
	xMsg1043.AmmOutAdr	:=  iAdrMM2AmmBase;

	xMsg1051.Num		:=	1051;
	xMsg1051.AmmInAdr	:=  iAdrAmmBase2MM;
	xMsg1051.AmmOutAdr	:=  iAdrMM2AmmBase;

	xMsg1052.Num		:=  1052;
	xMsg1052.AmmInAdr	:=  iAdrAmmBase2MM;
	xMsg1052.AmmOutAdr	:=  iAdrMM2AmmBase;

	xMsg1053.Num		:=  1053;
	xMsg1053.AmmInAdr	:=  iAdrAmmBase2MM;
	xMsg1053.AmmOutAdr	:=  iAdrMM2AmmBase;

	xMsg1054.Num		:=  1054;
	xMsg1054.AmmInAdr	:=  iAdrAmmBase2MM;
	xMsg1054.AmmOutAdr	:=  iAdrMM2AmmBase;

	xMsg1059.Num		:=	1059;
	xMsg1059.AmmInAdr	:=  iAdrAmmBase2MM;
	xMsg1059.AmmOutAdr	:=  iAdrMM2AmmBase;

	xMsg1060.Num		:=  1060;
	xMsg1060.AmmInAdr	:=  iAdrAmmBase2MM;
	xMsg1060.AmmOutAdr	:=  iAdrMM2AmmBase;

	xMsg1090.Num		:=  1090;
	xMsg1090.AmmInAdr	:=  iAdrAmmBase2MM;
	xMsg1090.AmmOutAdr	:=  iAdrMM2AmmBase;

	xMsg1091.Num		:=  1091;
	xMsg1091.AmmInAdr	:=  iAdrAmmBase2MM;
	xMsg1091.AmmOutAdr	:=  iAdrMM2AmmBase;

	xMsg1100.Num		:=  1100;
	xMsg1100.AmmInAdr	:=  iAdrAmmBase2MM;
	xMsg1100.AmmOutAdr	:=  iAdrMM2AmmBase;

	xMsg1101.Num		:=  1101;
	xMsg1101.AmmInAdr	:=  iAdrAmmBase2MM;
	xMsg1101.AmmOutAdr	:=  iAdrMM2AmmBase;

	xMsg1120.Num		:=  1120;
	xMsg1120.AmmInAdr	:=  iAdrAmmBase2MM;
	xMsg1120.AmmOutAdr	:=  iAdrMM2AmmBase;

	xMsg1129.Num		:=  1129;
	xMsg1129.AmmInAdr	:=  iAdrAmmBase2MM;
	xMsg1129.AmmOutAdr	:=  iAdrMM2AmmBase;

	xMsg1137.Num		:=  1137;
	xMsg1137.AmmInAdr	:=  iAdrAmmBase2MM;
	xMsg1137.AmmOutAdr	:=  iAdrMM2AmmBase;

	xMsg1139.Num		:=  1139;
	xMsg1139.AmmInAdr	:=  iAdrAmmBase2MM;
	xMsg1139.AmmOutAdr	:=  iAdrMM2AmmBase;

	xMsg1140.Num		:=  1140;
	xMsg1140.AmmInAdr	:=  iAdrAmmBase2MM;
	xMsg1140.AmmOutAdr	:=  iAdrMM2AmmBase;

	xMsg1148.Num		:=  1148;
	xMsg1148.AmmInAdr	:=  iAdrAmmBase2MM;
	xMsg1148.AmmOutAdr	:=  iAdrMM2AmmBase;

	xMsg1159.Num		:=  1159;
	xMsg1159.AmmInAdr	:=  iAdrAmmBase2MM;
	xMsg1159.AmmOutAdr	:=  iAdrMM2AmmBase;

	xMsg1160.Num		:=  1160;
	xMsg1160.AmmInAdr	:=  iAdrAmmBase2MM;
	xMsg1160.AmmOutAdr	:=  iAdrMM2AmmBase;

	xMsg1166.Num		:=	1166;
	xMsg1166.AmmInAdr	:=  iAdrAmmBase2MM;
	xMsg1166.AmmOutAdr	:=  iAdrMM2AmmBase;

	xMsg1249.Num		:=	1249;
	xMsg1249.AmmInAdr	:=  iAdrAmmBase2MM;
	xMsg1249.AmmOutAdr	:=  iAdrMM2AmmBase;

	xMsg1250.Num		:=	1250;
	xMsg1250.AmmInAdr	:=  iAdrAmmBase2MM;
	xMsg1250.AmmOutAdr	:=  iAdrMM2AmmBase;

	xMsg1257.Num		:=	1257;
	xMsg1257.AmmInAdr	:=  iAdrAmmBase2MM;
	xMsg1257.AmmOutAdr	:=  iAdrMM2AmmBase;

	xMsg1258.Num		:=	1258;
	xMsg1258.AmmInAdr	:=  iAdrAmmBase2MM;
	xMsg1258.AmmOutAdr	:=  iAdrMM2AmmBase;

	xMsg1259.Num		:=	1259;
	xMsg1259.AmmInAdr	:=  iAdrAmmBase2MM;
	xMsg1259.AmmOutAdr	:=  iAdrMM2AmmBase;

	xMsg1260.Num		:=	1260;
	xMsg1260.AmmInAdr	:=  iAdrAmmBase2MM;
	xMsg1260.AmmOutAdr	:=  iAdrMM2AmmBase;

	xMsg1261.Num		:=	1261;
	xMsg1261.AmmInAdr	:=  iAdrAmmBase2MM;
	xMsg1261.AmmOutAdr	:=  iAdrMM2AmmBase;

	xMsg1262.Num		:=	1262;
	xMsg1262.AmmInAdr	:=  iAdrAmmBase2MM;
	xMsg1262.AmmOutAdr	:=  iAdrMM2AmmBase;

	xMsg1263.Num		:=	1263;
	xMsg1263.AmmInAdr	:=  iAdrAmmBase2MM;
	xMsg1263.AmmOutAdr	:=  iAdrMM2AmmBase;

	xMsg1264.Num		:=	1264;
	xMsg1264.AmmInAdr	:=  iAdrAmmBase2MM;
	xMsg1264.AmmOutAdr	:=  iAdrMM2AmmBase;

	xMsg1281.Num		:=	1281;
	xMsg1281.AmmInAdr	:=  iAdrAmmBase2MM;
	xMsg1281.AmmOutAdr	:=  iAdrMM2AmmBase;

	xMsg1282.Num		:=	1282;
	xMsg1282.AmmInAdr	:=  iAdrAmmBase2MM;
	xMsg1282.AmmOutAdr	:=  iAdrMM2AmmBase;

	xMsg1292.Num		:=	1292;
	xMsg1292.AmmInAdr	:=  iAdrAmmBase2MM;
	xMsg1292.AmmOutAdr	:=  iAdrMM2AmmBase;

	xMsg2102.Num		:=	2102;
	xMsg2102.AmmInAdr	:=  iAdrAmmBase2MM;
	xMsg2102.AmmOutAdr	:=  iAdrMM2AmmBase;

	xMsg2103.Num		:=	2103;
	xMsg2103.AmmInAdr	:=  iAdrAmmBase2MM;
	xMsg2103.AmmOutAdr	:=  iAdrMM2AmmBase;

	xMsg2114.Num		:=  2114;
	xMsg2114.AmmInAdr	:=  iAdrAmmBase2MM;
	xMsg2114.AmmOutAdr	:=  iAdrMM2AmmBase;

	xMsg2118.Num		:=  2118;
	xMsg2118.AmmInAdr	:=  iAdrAmmBase2MM;
	xMsg2118.AmmOutAdr	:=  iAdrMM2AmmBase;

	xMsg2201.Num		:=  2201;
	xMsg2201.AmmInAdr	:=  iAdrAmmBase2MM;
	xMsg2201.AmmOutAdr	:=  iAdrMM2AmmBase;

	xMsg2213.Num		:=	2213;
	xMsg2213.AmmInAdr	:=  iAdrAmmBase2MM;
	xMsg2213.AmmOutAdr	:=  iAdrMM2AmmBase;

	xMsg2224.Num		:=	2224;
	xMsg2224.AmmInAdr	:=  iAdrAmmBase2MM;
	xMsg2224.AmmOutAdr	:=  iAdrMM2AmmBase;

	xMsg2233.Num		:=	2233;
	xMsg2233.AmmInAdr	:=  iAdrAmmBase2MM;
	xMsg2233.AmmOutAdr	:=  iAdrMM2AmmBase;

	xMsg2234.Num		:=	2234;
	xMsg2234.AmmInAdr	:=  iAdrAmmBase2MM;
	xMsg2234.AmmOutAdr	:=  iAdrMM2AmmBase;

	xMsg2238.Num		:=	2238;
	xMsg2238.AmmInAdr	:=  iAdrAmmBase2MM;
	xMsg2238.AmmOutAdr	:=  iAdrMM2AmmBase;

	xMsg2242.Num		:=	2242;
	xMsg2242.AmmInAdr	:=  iAdrAmmBase2MM;
	xMsg2242.AmmOutAdr	:=  iAdrMM2AmmBase;

	xMsg2260.Num		:=	2260;
	xMsg2260.AmmInAdr	:=  iAdrAmmBase2MM;
	xMsg2260.AmmOutAdr	:=  iAdrMM2AmmBase;

	xMsg2263.Num		:=  2263;
	xMsg2263.AmmInAdr	:=  iAdrAmmBase2MM;
	xMsg2263.AmmOutAdr	:=  iAdrMM2AmmBase;

	xMsg2264.Num		:=  2264;
	xMsg2264.AmmInAdr	:=  iAdrAmmBase2MM;
	xMsg2264.AmmOutAdr	:=  iAdrMM2AmmBase;

	xMsg2265.Num		:=  2265;
	xMsg2265.AmmInAdr	:=  iAdrAmmBase2MM;
	xMsg2265.AmmOutAdr	:=  iAdrMM2AmmBase;

	xMsg2266.Num		:=  2266;
	xMsg2266.AmmInAdr	:=  iAdrAmmBase2MM;
	xMsg2266.AmmOutAdr	:=  iAdrMM2AmmBase;

	xMsg2267.Num		:=  2267;
	xMsg2267.AmmInAdr	:=  iAdrAmmBase2MM;
	xMsg2267.AmmOutAdr	:=  iAdrMM2AmmBase;

	xMsg2268.Num		:=  2268;
	xMsg2268.AmmInAdr	:=  iAdrAmmBase2MM;
	xMsg2268.AmmOutAdr	:=  iAdrMM2AmmBase;

	xMsg2269.Num		:=  2269;
	xMsg2269.AmmInAdr	:=  iAdrAmmBase2MM;
	xMsg2269.AmmOutAdr	:=  iAdrMM2AmmBase;

	xMsg2284.Num		:=	2284;
	xMsg2284.AmmInAdr	:=  iAdrAmmBase2MM;
	xMsg2284.AmmOutAdr	:=  iAdrMM2AmmBase;

	xMsg2291.Num		:=  2291;
	xMsg2291.AmmInAdr	:=  iAdrAmmBase2MM;
	xMsg2291.AmmOutAdr	:=  iAdrMM2AmmBase;

	xMsg2292.Num		:=  2292;
	xMsg2292.AmmInAdr	:=  iAdrAmmBase2MM;
	xMsg2292.AmmOutAdr	:=  iAdrMM2AmmBase;

	xMsg2304.Num		:=	2304;
	xMsg2304.AmmInAdr	:=  iAdrAmmBase2MM;
	xMsg2304.AmmOutAdr	:=  iAdrMM2AmmBase;

	xMsg2332.Num		:=	2332;
	xMsg2332.AmmInAdr	:=  iAdrAmmBase2MM;
	xMsg2332.AmmOutAdr	:=  iAdrMM2AmmBase;

	xMsg2333.Num		:=	2333;
	xMsg2333.AmmInAdr	:=  iAdrAmmBase2MM;
	xMsg2333.AmmOutAdr	:=  iAdrMM2AmmBase;

	xMsg2348.Num		:=	2348;
	xMsg2348.AmmInAdr	:=  iAdrAmmBase2MM;
	xMsg2348.AmmOutAdr	:=  iAdrMM2AmmBase;

	xMsg2349.Num		:=	2349;
	xMsg2349.AmmInAdr	:=  iAdrAmmBase2MM;
	xMsg2349.AmmOutAdr	:=  iAdrMM2AmmBase;

	xMsg2350.Num		:=	2350;
	xMsg2350.AmmInAdr	:=  iAdrAmmBase2MM;
	xMsg2350.AmmOutAdr	:=  iAdrMM2AmmBase;

	xMsg2351.Num		:=	2351;
	xMsg2351.AmmInAdr	:=  iAdrAmmBase2MM;
	xMsg2351.AmmOutAdr	:=  iAdrMM2AmmBase;

	xMsg2352.Num		:=	2352;
	xMsg2352.AmmInAdr	:=  iAdrAmmBase2MM;
	xMsg2352.AmmOutAdr	:=  iAdrMM2AmmBase;

	xMsg2353.Num		:=	2353;
	xMsg2353.AmmInAdr	:=  iAdrAmmBase2MM;
	xMsg2353.AmmOutAdr	:=  iAdrMM2AmmBase;

	xMsg2355.Num		:=	2355;
	xMsg2355.AmmInAdr	:=  iAdrAmmBase2MM;
	xMsg2355.AmmOutAdr	:=  iAdrMM2AmmBase;

	xMsg2359.Num		:=	2359;
	xMsg2359.AmmInAdr	:=  iAdrAmmBase2MM;
	xMsg2359.AmmOutAdr	:=  iAdrMM2AmmBase;

	xMsg2360.Num		:=	2360;
	xMsg2360.AmmInAdr	:=  iAdrAmmBase2MM;
	xMsg2360.AmmOutAdr	:=  iAdrMM2AmmBase;

	xMsg2361.Num		:=	2361;
	xMsg2361.AmmInAdr	:=  iAdrAmmBase2MM;
	xMsg2361.AmmOutAdr	:=  iAdrMM2AmmBase;

	xMsg2376.Num		:=	2376;
	xMsg2376.AmmInAdr	:=  iAdrAmmBase2MM;
	xMsg2376.AmmOutAdr	:=  iAdrMM2AmmBase;

	xMsg2377.Num		:=	2377;
	xMsg2377.AmmInAdr	:=  iAdrAmmBase2MM;
	xMsg2377.AmmOutAdr	:=  iAdrMM2AmmBase;

	xMsg2378.Num		:=	2378;
	xMsg2378.AmmInAdr	:=  iAdrAmmBase2MM;
	xMsg2378.AmmOutAdr	:=  iAdrMM2AmmBase;

	xMsg2379.Num		:=	2379;
	xMsg2379.AmmInAdr	:=  iAdrAmmBase2MM;
	xMsg2379.AmmOutAdr	:=  iAdrMM2AmmBase;

	xMsg2382.Num		:=	2382;
	xMsg2382.AmmInAdr	:=  iAdrAmmBase2MM;
	xMsg2382.AmmOutAdr	:=  iAdrMM2AmmBase;

	xMsg2421.Num		:=	2421;
	xMsg2421.AmmInAdr	:=  iAdrAmmBase2MM;
	xMsg2421.AmmOutAdr	:=  iAdrMM2AmmBase;

	xMsg2422.Num		:=  2422;
	xMsg2422.AmmInAdr	:=  iAdrAmmBase2MM;
	xMsg2422.AmmOutAdr	:=  iAdrMM2AmmBase;

	xMsg2423.Num		:=	2423;//SWAT920/1
	xMsg2423.AmmInAdr	:=  iAdrAmmBase2MM;
	xMsg2423.AmmOutAdr	:=  iAdrMM2AmmBase;

	xMsg2424.Num		:=	2424;//SWAT920/2.2
	xMsg2424.AmmInAdr	:=  iAdrAmmBase2MM;
	xMsg2424.AmmOutAdr	:=  iAdrMM2AmmBase;

	xMsg2425.Num		:=	2425;//SWAT920/2.2
	xMsg2425.AmmInAdr	:=  iAdrAmmBase2MM;
	xMsg2425.AmmOutAdr	:=  iAdrMM2AmmBase;

	xMsg2426.Num		:=	2426;//SWAT920/2.2
	xMsg2426.AmmInAdr	:=  iAdrAmmBase2MM;
	xMsg2426.AmmOutAdr	:=  iAdrMM2AmmBase;

	xMsg2427.Num		:=	2427;
	xMsg2427.AmmInAdr	:=  iAdrAmmBase2MM;
	xMsg2427.AmmOutAdr	:=  iAdrMM2AmmBase;

	xMsg2431.Num		:=	2431;//SWAT920/1
	xMsg2431.AmmInAdr	:=  iAdrAmmBase2MM;
	xMsg2431.AmmOutAdr	:=  iAdrMM2AmmBase;

	xMsg2432.Num		:=	2432;//SWAT920/1
	xMsg2432.AmmInAdr	:=  iAdrAmmBase2MM;
	xMsg2432.AmmOutAdr	:=  iAdrMM2AmmBase;

	xMsg2433.Num		:=	2433;//SWAT920/1
	xMsg2433.AmmInAdr	:=  iAdrAmmBase2MM;
	xMsg2433.AmmOutAdr	:=  iAdrMM2AmmBase;

	xMsg2434.Num		:=	2434;
	xMsg2434.AmmInAdr	:=  iAdrAmmBase2MM;
	xMsg2434.AmmOutAdr	:=  iAdrMM2AmmBase;

	xMsg2435.Num		:=	2435;//SWAT920/2
	xMsg2435.AmmInAdr	:=  iAdrAmmBase2MM;
	xMsg2435.AmmOutAdr	:=  iAdrMM2AmmBase;

	xMsg2459.Num		:=  2459;
	xMsg2459.AmmInAdr	:=  iAdrAmmBase2MM;
	xMsg2459.AmmOutAdr	:=  iAdrMM2AmmBase;

	xMsg2473.Num		:=  2473;
	xMsg2473.AmmInAdr	:=  iAdrAmmBase2MM;
	xMsg2473.AmmOutAdr	:=  iAdrMM2AmmBase;

	xMsg2475.Num		:=  2475;
	xMsg2475.AmmInAdr	:=  iAdrAmmBase2MM;
	xMsg2475.AmmOutAdr	:=  iAdrMM2AmmBase;

	xMsg2524.Num		:=	2524;
	xMsg2524.AmmInAdr	:=  iAdrAmmBase2MM;
	xMsg2524.AmmOutAdr	:=  iAdrMM2AmmBase;

	xMsg2534.Num		:=	2534;
	xMsg2534.AmmInAdr	:=  iAdrAmmBase2MM;
	xMsg2534.AmmOutAdr	:=  iAdrMM2AmmBase;

	xMsg2545.Num		:=  2545;
	xMsg2545.AmmInAdr	:=  iAdrAmmBase2MM;
	xMsg2545.AmmOutAdr	:=  iAdrMM2AmmBase;

	xMsg2554.Num		:=	2554;
	xMsg2554.AmmInAdr	:=  iAdrAmmBase2MM;
	xMsg2554.AmmOutAdr	:=  iAdrMM2AmmBase;

	xMsg2557.Num		:=	2557;//SWAT920/2.2
	xMsg2557.AmmInAdr	:=  iAdrAmmBase2MM;
	xMsg2557.AmmOutAdr	:=  iAdrMM2AmmBase;

	xMsg2558.Num		:=  2558;
	xMsg2558.AmmInAdr	:=  iAdrAmmBase2MM;
	xMsg2558.AmmOutAdr	:=  iAdrMM2AmmBase;

	xMsg2559.Num 		:=  2559;
	xMsg2559.AmmInAdr 	:=  iAdrAmmBase2MM;
	xMsg2559.AmmOutAdr 	:=  iAdrMM2AmmBase;

	xMsg2560.Num		:=  2560;
	xMsg2560.AmmInAdr	:=  iAdrAmmBase2MM;
	xMsg2560.AmmOutAdr	:=  iAdrMM2AmmBase;

	xMsg2571.Num		:=  2571;
	xMsg2571.AmmInAdr	:=  iAdrAmmBase2MM;
	xMsg2571.AmmOutAdr	:=  iAdrMM2AmmBase;

	xMsg2572.Num		:=  2572;
	xMsg2572.AmmInAdr	:=  iAdrAmmBase2MM;
	xMsg2572.AmmOutAdr	:=  iAdrMM2AmmBase;

	xMsg2576.Num		:=	2576;
	xMsg2576.AmmInAdr	:=  iAdrAmmBase2MM;
	xMsg2576.AmmOutAdr	:=  iAdrMM2AmmBase;

	xMsg2579.Num		:=	2579;
	xMsg2579.AmmInAdr	:=  iAdrAmmBase2MM;
	xMsg2579.AmmOutAdr	:=  iAdrMM2AmmBase;

	xMsg2582.Num		:=	2582;
	xMsg2582.AmmInAdr	:=  iAdrAmmBase2MM;
	xMsg2582.AmmOutAdr	:=  iAdrMM2AmmBase;

	xMsg2587.Num		:=	2587;
	xMsg2587.AmmInAdr	:=  iAdrAmmBase2MM;
	xMsg2587.AmmOutAdr	:=  iAdrMM2AmmBase;

	xMsg2589.Num		:=  2589;
	xMsg2589.AmmInAdr	:=  iAdrAmmBase2MM;
	xMsg2589.AmmOutAdr	:=  iAdrMM2AmmBase;

	xMsg2590.Num		:=  2590;
	xMsg2590.AmmInAdr	:=  iAdrAmmBase2MM;
	xMsg2590.AmmOutAdr	:=  iAdrMM2AmmBase;

	xMsg2591.Num		:=  2591;
	xMsg2591.AmmInAdr	:=  iAdrAmmBase2MM;
	xMsg2591.AmmOutAdr	:=  iAdrMM2AmmBase;

	xMsg2592.Num		:=  2592;
	xMsg2592.AmmInAdr	:=  iAdrAmmBase2MM;
	xMsg2592.AmmOutAdr	:=  iAdrMM2AmmBase;

	xMsg2594.Num		:=  2594;
	xMsg2594.AmmInAdr	:=  iAdrAmmBase2MM;
	xMsg2594.AmmOutAdr	:=  iAdrMM2AmmBase;

	xMsg2595.Num		:=  2595;
	xMsg2595.AmmInAdr	:=  iAdrAmmBase2MM;
	xMsg2595.AmmOutAdr	:=  iAdrMM2AmmBase;

	xMsg2596.Num		:=  2596;
	xMsg2596.AmmInAdr	:=  iAdrAmmBase2MM;
	xMsg2596.AmmOutAdr	:=  iAdrMM2AmmBase;

	xMsg2597.Num		:=	2597;
	xMsg2597.AmmInAdr	:=  iAdrAmmBase2MM;
	xMsg2597.AmmOutAdr	:=  iAdrMM2AmmBase;

	xMsg2598.Num		:=	2598;
	xMsg2598.AmmInAdr	:=  iAdrAmmBase2MM;
	xMsg2598.AmmOutAdr	:=  iAdrMM2AmmBase;

	xMsg2599.Num		:=	2599;
	xMsg2599.AmmInAdr	:=  iAdrAmmBase2MM;
	xMsg2599.AmmOutAdr	:=  iAdrMM2AmmBase;

	xMsg2600.Num		:=	2600;
	xMsg2600.AmmInAdr	:=  iAdrAmmBase2MM;
	xMsg2600.AmmOutAdr	:=  iAdrMM2AmmBase;

	xMsg2602.Num		:=	2602;
	xMsg2602.AmmInAdr	:=  iAdrAmmBase2MM;
	xMsg2602.AmmOutAdr	:=  iAdrMM2AmmBase;

	xMsg2603.Num		:=	2603;
	xMsg2603.AmmInAdr	:=  iAdrAmmBase2MM;
	xMsg2603.AmmOutAdr	:=  iAdrMM2AmmBase;

	xMsg2604.Num		:=	2604;
	xMsg2604.AmmInAdr	:=  iAdrAmmBase2MM;
	xMsg2604.AmmOutAdr	:=  iAdrMM2AmmBase;

	xMsg2605.Num		:=	2605;
	xMsg2605.AmmInAdr	:=  iAdrAmmBase2MM;
	xMsg2605.AmmOutAdr	:=  iAdrMM2AmmBase;

	xMsg2606.Num		:=	2606;
	xMsg2606.AmmInAdr	:=  iAdrAmmBase2MM;
	xMsg2606.AmmOutAdr	:=  iAdrMM2AmmBase;

	xMsg2608.Num		:=	2608;
	xMsg2608.AmmInAdr	:=  iAdrAmmBase2MM;
	xMsg2608.AmmOutAdr	:=  iAdrMM2AmmBase;

	xMsg2613.Num		:=	2613;
	xMsg2613.AmmInAdr	:=  iAdrAmmBase2MM;
	xMsg2613.AmmOutAdr	:=  iAdrMM2AmmBase;

	xMsg2624.Num		:=	2624;
	xMsg2624.AmmInAdr	:=  iAdrAmmBase2MM;
	xMsg2624.AmmOutAdr	:=  iAdrMM2AmmBase;

	xMsg2625.Num		:=	2625;
	xMsg2625.AmmInAdr	:=  iAdrAmmBase2MM;
	xMsg2625.AmmOutAdr	:=  iAdrMM2AmmBase;

	xMsg2627.Num		:=	2627;
	xMsg2627.AmmInAdr	:=  iAdrAmmBase2MM;
	xMsg2627.AmmOutAdr	:=  iAdrMM2AmmBase;

	xMsg2628.Num		:=	2628;
	xMsg2628.AmmInAdr	:=  iAdrAmmBase2MM;
	xMsg2628.AmmOutAdr	:=  iAdrMM2AmmBase;

	xMsg2629.Num		:=	2629;
	xMsg2629.AmmInAdr	:=  iAdrAmmBase2MM;
	xMsg2629.AmmOutAdr	:=  iAdrMM2AmmBase;

	xMsg2636.Num		:=	2636;
	xMsg2636.AmmInAdr	:=  iAdrAmmBase2MM;
	xMsg2636.AmmOutAdr	:=  iAdrMM2AmmBase;

	xMsg2642.Num		:=	2642;
	xMsg2642.AmmInAdr	:=  iAdrAmmBase2MM;
	xMsg2642.AmmOutAdr	:=  iAdrMM2AmmBase;

	xMsg2643.Num		:=	2643;
	xMsg2643.AmmInAdr	:=  iAdrAmmBase2MM;
	xMsg2643.AmmOutAdr	:=  iAdrMM2AmmBase;

	xMsg2644.Num		:=	2644;
	xMsg2644.AmmInAdr	:=  iAdrAmmBase2MM;
	xMsg2644.AmmOutAdr	:=  iAdrMM2AmmBase;

	xMsg2645.Num		:=	2645;
	xMsg2645.AmmInAdr	:=  iAdrAmmBase2MM;
	xMsg2645.AmmOutAdr	:=  iAdrMM2AmmBase;

	xMsg2646.Num		:=	2646;
	xMsg2646.AmmInAdr	:=  iAdrAmmBase2MM;
	xMsg2646.AmmOutAdr	:=  iAdrMM2AmmBase;

	xMsg2648.Num		:=	2648;
	xMsg2648.AmmInAdr	:=  iAdrAmmBase2MM;
	xMsg2648.AmmOutAdr	:=  iAdrMM2AmmBase;

	xMsg2649.Num 		:= 	2649;
	xMsg2649.AmmInAdr 	:= iAdrAmmBase2MM;
	xMsg2649.AmmOutAdr 	:= iAdrMM2AmmBase;

	xMsg2650.Num 		:= 	2650;
	xMsg2650.AmmInAdr 	:= iAdrAmmBase2MM;
	xMsg2650.AmmOutAdr 	:= iAdrMM2AmmBase;

	xMsg2651.Num 		:= 	2651;
	xMsg2651.AmmInAdr 	:= iAdrAmmBase2MM;
	xMsg2651.AmmOutAdr 	:= iAdrMM2AmmBase;

	xMsg2652.Num 		:= 	2652;
	xMsg2652.AmmInAdr 	:= iAdrAmmBase2MM;
	xMsg2652.AmmOutAdr 	:= iAdrMM2AmmBase;

	xMsg2653.Num 		:= 	2653;
	xMsg2653.AmmInAdr 	:= iAdrAmmBase2MM;
	xMsg2653.AmmOutAdr 	:= iAdrMM2AmmBase;

	xMsg2654.Num 		:= 	2654;
	xMsg2654.AmmInAdr 	:= iAdrAmmBase2MM;
	xMsg2654.AmmOutAdr 	:= iAdrMM2AmmBase;

	xMsg2666.Num		:=	2666;
	xMsg2666.AmmInAdr	:=  iAdrAmmBase2MM;
	xMsg2666.AmmOutAdr	:=  iAdrMM2AmmBase;

	xMsg2689.Num		:=	2689;
	xMsg2689.AmmInAdr	:=  iAdrAmmBase2MM;
	xMsg2689.AmmOutAdr	:=  iAdrMM2AmmBase;

	xMsg2722.Num		:=	2722;
	xMsg2722.AmmInAdr	:=  iAdrAmmBase2MM;
	xMsg2722.AmmOutAdr	:=  iAdrMM2AmmBase;

	xMsg2723.Num		:=	2723;
	xMsg2723.AmmInAdr	:=  iAdrAmmBase2MM;
	xMsg2723.AmmOutAdr	:=  iAdrMM2AmmBase;

	xMsg2724.Num		:=	2724;
	xMsg2724.AmmInAdr	:=  iAdrAmmBase2MM;
	xMsg2724.AmmOutAdr	:=  iAdrMM2AmmBase;

	xMsg2725.Num		:=	2725;
	xMsg2725.AmmInAdr	:=  iAdrAmmBase2MM;
	xMsg2725.AmmOutAdr	:=  iAdrMM2AmmBase;

	xMsg2726.Num		:=	2726;
	xMsg2726.AmmInAdr	:=  iAdrAmmBase2MM;
	xMsg2726.AmmOutAdr	:=  iAdrMM2AmmBase;

	xMsg2727.Num		:=	2727;
	xMsg2727.AmmInAdr	:=  iAdrAmmBase2MM;
	xMsg2727.AmmOutAdr	:=  iAdrMM2AmmBase;

	xMsg2728.Num		:=	2728;
	xMsg2728.AmmInAdr	:=  iAdrAmmBase2MM;
	xMsg2728.AmmOutAdr	:=  iAdrMM2AmmBase;

	xMsg2729.Num		:=	2729;
	xMsg2729.AmmInAdr	:=  iAdrAmmBase2MM;
	xMsg2729.AmmOutAdr	:=  iAdrMM2AmmBase;

	xMsg2737.Num		:=	2737;
	xMsg2737.AmmInAdr	:=  iAdrAmmBase2MM;
	xMsg2737.AmmOutAdr	:=  iAdrMM2AmmBase;

	xMsg2738.Num		:=	2738;
	xMsg2738.AmmInAdr	:=  iAdrAmmBase2MM;
	xMsg2738.AmmOutAdr	:=  iAdrMM2AmmBase;

	xMsg2739.Num		:=	2739;
	xMsg2739.AmmInAdr	:=  iAdrAmmBase2MM;
	xMsg2739.AmmOutAdr	:=  iAdrMM2AmmBase;

	xMsg2740.Num		:=	2740;
	xMsg2740.AmmInAdr	:=  iAdrAmmBase2MM;
	xMsg2740.AmmOutAdr	:=  iAdrMM2AmmBase;

	xMsg2741.Num		:=	2741;
	xMsg2741.AmmInAdr	:=  iAdrAmmBase2MM;
	xMsg2741.AmmOutAdr	:=  iAdrMM2AmmBase;

	xMsg2742.Num		:=	2742;
	xMsg2742.AmmInAdr	:=  iAdrAmmBase2MM;
	xMsg2742.AmmOutAdr	:=  iAdrMM2AmmBase;

	xMsg2754.Num		:=	2754;
	xMsg2754.AmmInAdr	:=  iAdrAmmBase2MM;
	xMsg2754.AmmOutAdr	:=  iAdrMM2AmmBase;

	xMsg2755.Num		:=	2755;
	xMsg2755.AmmInAdr	:=  iAdrAmmBase2MM;
	xMsg2755.AmmOutAdr	:=  iAdrMM2AmmBase;

	xMsg2756.Num		:=	2756;
	xMsg2756.AmmInAdr	:=  iAdrAmmBase2MM;
	xMsg2756.AmmOutAdr	:=  iAdrMM2AmmBase;

	xMsg2757.Num		:=	2757;
	xMsg2757.AmmInAdr	:=  iAdrAmmBase2MM;
	xMsg2757.AmmOutAdr	:=  iAdrMM2AmmBase;

	xMsg2758.Num		:=	2758;
	xMsg2758.AmmInAdr	:=  iAdrAmmBase2MM;
	xMsg2758.AmmOutAdr	:=  iAdrMM2AmmBase;

	xMsg2759.Num		:=	2759;
	xMsg2759.AmmInAdr	:=  iAdrAmmBase2MM;
	xMsg2759.AmmOutAdr	:=  iAdrMM2AmmBase;

	xMsg2760.Num		:=	2760;
	xMsg2760.AmmInAdr	:=  iAdrAmmBase2MM;
	xMsg2760.AmmOutAdr	:=  iAdrMM2AmmBase;

	xMsg2761.Num		:=	2761;
	xMsg2761.AmmInAdr	:=  iAdrAmmBase2MM;
	xMsg2761.AmmOutAdr	:=  iAdrMM2AmmBase;

	xMsg2762.Num		:=	2762;
	xMsg2762.AmmInAdr	:=  iAdrAmmBase2MM;
	xMsg2762.AmmOutAdr	:=  iAdrMM2AmmBase;

	xMsg2770.Num		:=	2770;
	xMsg2770.AmmInAdr	:=  iAdrAmmBase2MM;
	xMsg2770.AmmOutAdr	:=  iAdrMM2AmmBase;

	xMsg2771.Num		:=	2771;
	xMsg2771.AmmInAdr	:=  iAdrAmmBase2MM;
	xMsg2771.AmmOutAdr	:=  iAdrMM2AmmBase;

	xMsg2772.Num		:=	2772;
	xMsg2772.AmmInAdr	:=  iAdrAmmBase2MM;
	xMsg2772.AmmOutAdr	:=  iAdrMM2AmmBase;

	xMsg2773.Num		:=	2773;
	xMsg2773.AmmInAdr	:=  iAdrAmmBase2MM;
	xMsg2773.AmmOutAdr	:=  iAdrMM2AmmBase;

	xMsg2774.Num		:=	2774;
	xMsg2774.AmmInAdr	:=  iAdrAmmBase2MM;
	xMsg2774.AmmOutAdr	:=  iAdrMM2AmmBase;

	xMsg2775.Num		:=	2775;
	xMsg2775.AmmInAdr	:=  iAdrAmmBase2MM;
	xMsg2775.AmmOutAdr	:=  iAdrMM2AmmBase;

	xMsg2776.Num		:=	2776;
	xMsg2776.AmmInAdr	:=  iAdrAmmBase2MM;
	xMsg2776.AmmOutAdr	:=  iAdrMM2AmmBase;

	xMsg2777.Num		:=	2777;
	xMsg2777.AmmInAdr	:=  iAdrAmmBase2MM;
	xMsg2777.AmmOutAdr	:=  iAdrMM2AmmBase;

	xMsg2778.Num		:=	2778;
	xMsg2778.AmmInAdr	:=  iAdrAmmBase2MM;
	xMsg2778.AmmOutAdr	:=  iAdrMM2AmmBase;

	xMsg2781.Num		:=	2781;
	xMsg2781.AmmInAdr	:=  iAdrAmmBase2MM;
	xMsg2781.AmmOutAdr	:=  iAdrMM2AmmBase;

	xMsg2782.Num		:=	2782;
	xMsg2782.AmmInAdr	:=  iAdrAmmBase2MM;
	xMsg2782.AmmOutAdr	:=  iAdrMM2AmmBase;

	xMsg2783.Num		:=	2783;
	xMsg2783.AmmInAdr	:=  iAdrAmmBase2MM;
	xMsg2783.AmmOutAdr	:=  iAdrMM2AmmBase;

	xMsg2784.Num		:=	2784;
	xMsg2784.AmmInAdr	:=  iAdrAmmBase2MM;
	xMsg2784.AmmOutAdr	:=  iAdrMM2AmmBase;

	xMsg2785.Num		:=	2785;
	xMsg2785.AmmInAdr	:=  iAdrAmmBase2MM;
	xMsg2785.AmmOutAdr	:=  iAdrMM2AmmBase;

	xMsg2786.Num		:=	2786;
	xMsg2786.AmmInAdr	:=  iAdrAmmBase2MM;
	xMsg2786.AmmOutAdr	:=  iAdrMM2AmmBase;

	xMsg2787.Num		:=	2787;
	xMsg2787.AmmInAdr	:=  iAdrAmmBase2MM;
	xMsg2787.AmmOutAdr	:=  iAdrMM2AmmBase;

	xMsg2788.Num		:=	2788;
	xMsg2788.AmmInAdr	:=  iAdrAmmBase2MM;
	xMsg2788.AmmOutAdr	:=  iAdrMM2AmmBase;

	xMsg2789.Num		:=	2789;
	xMsg2789.AmmInAdr	:=  iAdrAmmBase2MM;
	xMsg2789.AmmOutAdr	:=  iAdrMM2AmmBase;

	xMsg2791.Num		:=	2791;
	xMsg2791.AmmInAdr	:=  iAdrAmmBase2MM;
	xMsg2791.AmmOutAdr	:=  iAdrMM2AmmBase;

	xMsg2792.Num		:=	2792;
	xMsg2792.AmmInAdr	:=  iAdrAmmBase2MM;
	xMsg2792.AmmOutAdr	:=  iAdrMM2AmmBase;

	xMsg2809.Num		:=	2809;
	xMsg2809.AmmInAdr	:=  iAdrAmmBase2MM;
	xMsg2809.AmmOutAdr	:=  iAdrMM2AmmBase;

	xMsg2810.Num		:=	2810;
	xMsg2810.AmmInAdr	:=  iAdrAmmBase2MM;
	xMsg2810.AmmOutAdr	:=  iAdrMM2AmmBase;

	xMsg2931.Num		:=	2931;
	xMsg2931.AmmInAdr	:=  iAdrAmmBase2MM;
	xMsg2931.AmmOutAdr	:=  iAdrMM2AmmBase;

	xMsg2932.Num		:=	2932;
	xMsg2932.AmmInAdr	:=  iAdrAmmBase2MM;
	xMsg2932.AmmOutAdr	:=  iAdrMM2AmmBase;

	xMsg2933.Num		:=	2933;
	xMsg2933.AmmInAdr	:=  iAdrAmmBase2MM;
	xMsg2933.AmmOutAdr	:=  iAdrMM2AmmBase;

	xMsg2956.Num		:=	2956;
	xMsg2956.AmmInAdr	:=  iAdrAmmBase2MM;
	xMsg2956.AmmOutAdr	:=  iAdrMM2AmmBase;

	xMsg2957.Num		:=	2957;
	xMsg2957.AmmInAdr	:=  iAdrAmmBase2MM;
	xMsg2957.AmmOutAdr	:=  iAdrMM2AmmBase;

	xMsg2978.Num		:=	2978;
	xMsg2978.AmmInAdr	:=  iAdrAmmBase2MM;
	xMsg2978.AmmOutAdr	:=  iAdrMM2AmmBase;

	xMsg2979.Num		:=	2979;
	xMsg2979.AmmInAdr	:=  iAdrAmmBase2MM;
	xMsg2979.AmmOutAdr	:=  iAdrMM2AmmBase;

	xMsg3216.Num		:=	3216;
	xMsg3216.AmmInAdr	:=  iAdrAmmBase2MM;
	xMsg3216.AmmOutAdr	:=  iAdrMM2AmmBase;

	xMsg3218.Num		:=	3218;
	xMsg3218.AmmInAdr	:=  iAdrAmmBase2MM;
	xMsg3218.AmmOutAdr	:=  iAdrMM2AmmBase;

	xMsg3300.Num		:=	3300;
	xMsg3300.AmmInAdr	:=  iAdrAmmBase2MM;
	xMsg3300.AmmOutAdr	:=  iAdrMM2AmmBase;

	xMsg3301.Num		:=  3301;
	xMsg3301.AmmInAdr	:=  iAdrAmmBase2MM;
	xMsg3301.AmmOutAdr	:=  iAdrMM2AmmBase;

	xMsg3304.Num		:=	3304;
	xMsg3304.AmmInAdr	:=  iAdrAmmBase2MM;
	xMsg3304.AmmOutAdr	:=  iAdrMM2AmmBase;

	xMsg3305.Num		:=	3305;
	xMsg3305.AmmInAdr	:=  iAdrAmmBase2MM;
	xMsg3305.AmmOutAdr	:=  iAdrMM2AmmBase;

	xMsg3322.Num		:=  3322;
	xMsg3322.AmmInAdr	:=  iAdrAmmBase2MM;
	xMsg3322.AmmOutAdr	:=  iAdrMM2AmmBase;

	xMsg3323.Num		:=  3323;
	xMsg3323.AmmInAdr	:=  iAdrAmmBase2MM;
	xMsg3323.AmmOutAdr	:=  iAdrMM2AmmBase;

	xMsg3350.Num		:=  3350;
	xMsg3350.AmmInAdr	:=  iAdrAmmBase2MM;
	xMsg3350.AmmOutAdr	:=  iAdrMM2AmmBase;

	xMsg3351.Num		:=  3351;
	xMsg3351.AmmInAdr	:=  iAdrAmmBase2MM;
	xMsg3351.AmmOutAdr	:=  iAdrMM2AmmBase;

	xMsg3369.Num 		:= 3369;
	xMsg3369.AmmInAdr 	:= iAdrAmmBase2MM;
	xMsg3369.AmmOutAdr 	:= iAdrMM2AmmBase;

	xMsg3370.Num 		:= 3370;
	xMsg3370.AmmInAdr 	:= iAdrAmmBase2MM;
	xMsg3370.AmmOutAdr 	:= iAdrMM2AmmBase;

	xMsg3375.Num 		:= 3375;
	xMsg3375.AmmInAdr 	:= iAdrAmmBase2MM;
	xMsg3375.AmmOutAdr 	:= iAdrMM2AmmBase;

	xMsg3401.Num		:=  3401;
	xMsg3401.AmmInAdr	:=  iAdrAmmBase2MM;
	xMsg3401.AmmOutAdr	:=  iAdrMM2AmmBase;

	xMsg3403.Num		:=  3403;
	xMsg3403.AmmInAdr	:=  iAdrAmmBase2MM;
	xMsg3403.AmmOutAdr	:=  iAdrMM2AmmBase;

	xMsg3405.Num		:=  3405;
	xMsg3405.AmmInAdr	:=  iAdrAmmBase2MM;
	xMsg3405.AmmOutAdr	:=  iAdrMM2AmmBase;

	xMsg3413.Num		:=	3413;
	xMsg3413.AmmInAdr	:=  iAdrAmmBase2MM;
	xMsg3413.AmmOutAdr	:=  iAdrMM2AmmBase;

	xMsg3414.Num		:=	3414;
	xMsg3414.AmmInAdr	:=  iAdrAmmBase2MM;
	xMsg3414.AmmOutAdr	:=  iAdrMM2AmmBase;

	xMsg3415.Num		:=	3415;
	xMsg3415.AmmInAdr	:=  iAdrAmmBase2MM;
	xMsg3415.AmmOutAdr	:=  iAdrMM2AmmBase;

	xMsg3416.Num		:=	3416;
	xMsg3416.AmmInAdr	:=  iAdrAmmBase2MM;
	xMsg3416.AmmOutAdr	:=  iAdrMM2AmmBase;

	xMsg3495.Num		:=  3495;
	xMsg3495.AmmInAdr	:=  iAdrAmmBase2MM;
	xMsg3495.AmmOutAdr	:=  iAdrMM2AmmBase;

	xMsg3496.Num		:=  3496;
	xMsg3496.AmmInAdr	:=  iAdrAmmBase2MM;
	xMsg3496.AmmOutAdr	:=  iAdrMM2AmmBase;

	xMsg3497.Num		:=  3497;
	xMsg3497.AmmInAdr	:=  iAdrAmmBase2MM;
	xMsg3497.AmmOutAdr	:=  iAdrMM2AmmBase;

	xMsg3507.Num		:=	3507;
	xMsg3507.AmmInAdr	:=  iAdrAmmBase2MM;
	xMsg3507.AmmOutAdr	:=  iAdrMM2AmmBase;

	xMsg3515.Num		:=  3515;
	xMsg3515.AmmInAdr	:=  iAdrAmmBase2MM;
	xMsg3515.AmmOutAdr	:=  iAdrMM2AmmBase;

	xMsg3519.Num		:=  3519;
	xMsg3519.AmmInAdr	:=  iAdrAmmBase2MM;
	xMsg3519.AmmOutAdr	:=  iAdrMM2AmmBase;

	xMsg3572.Num		:=  3572;
	xMsg3572.AmmInAdr	:=  iAdrAmmBase2MM;
	xMsg3572.AmmOutAdr	:=  iAdrMM2AmmBase;

	xMsg3574.Num		:=  3574;
	xMsg3574.AmmInAdr	:=  iAdrAmmBase2MM;
	xMsg3574.AmmOutAdr	:=  iAdrMM2AmmBase;

	xMsg3578.Num		:=  3578;
	xMsg3578.AmmInAdr	:=  iAdrAmmBase2MM;
	xMsg3578.AmmOutAdr	:=  iAdrMM2AmmBase;

	xMsg3579.Num		:=  3579;
	xMsg3579.AmmInAdr	:=  iAdrAmmBase2MM;
	xMsg3579.AmmOutAdr	:=  iAdrMM2AmmBase;

	xMsg3587.Num		:=	3587;
	xMsg3587.AmmInAdr	:=  iAdrAmmBase2MM;
	xMsg3587.AmmOutAdr	:=  iAdrMM2AmmBase;

	xMsg3588.Num		:=	3588;
	xMsg3588.AmmInAdr	:=  iAdrAmmBase2MM;
	xMsg3588.AmmOutAdr	:=  iAdrMM2AmmBase;

	xMsg9001.Num		:=	9001;
	xMsg9001.AmmInAdr	:=  iAdrAmmBase2MM;
	xMsg9001.AmmOutAdr	:=  iAdrMM2AmmBase;

	xMsg9002.Num		:=	9002;
	xMsg9002.AmmInAdr	:=  iAdrAmmBase2MM;
	xMsg9002.AmmOutAdr	:=  iAdrMM2AmmBase;

	xMsg9003.Num		:=	9003;
	xMsg9003.AmmInAdr	:=  iAdrAmmBase2MM;
	xMsg9003.AmmOutAdr	:=  iAdrMM2AmmBase;

	xMsg9048.Num		:=	9048;
	xMsg9048.AmmInAdr	:=  iAdrAmmBase2MM;
	xMsg9048.AmmOutAdr	:=  iAdrMM2AmmBase;

	xMsg9067.Num		:=	9067;
	xMsg9067.AmmInAdr	:=  iAdrAmmBase2MM;
	xMsg9067.AmmOutAdr	:=  iAdrMM2AmmBase;

	xMsg9069.Num		:=	9069;
	xMsg9069.AmmInAdr	:=  iAdrAmmBase2MM;
	xMsg9069.AmmOutAdr	:=  iAdrMM2AmmBase;

	xMsg9070.Num		:=	9070;
	xMsg9070.AmmInAdr	:=  iAdrAmmBase2MM;
	xMsg9070.AmmOutAdr	:=  iAdrMM2AmmBase;

	xMsg9074.Num		:=	9074;
	xMsg9074.AmmInAdr	:=  iAdrAmmBase2MM;
	xMsg9074.AmmOutAdr	:=  iAdrMM2AmmBase;

	xMsg9088.Num		:=	9088;
	xMsg9088.AmmInAdr	:=  iAdrAmmBase2MM;
	xMsg9088.AmmOutAdr	:=  iAdrMM2AmmBase;

	xMsg9089.Num		:=	9089;
	xMsg9089.AmmInAdr	:=  iAdrAmmBase2MM;
	xMsg9089.AmmOutAdr	:=  iAdrMM2AmmBase;

	xMsg9090.Num		:=	9090;
	xMsg9090.AmmInAdr	:=  iAdrAmmBase2MM;
	xMsg9090.AmmOutAdr	:=  iAdrMM2AmmBase;

	xMsg9091.Num		:=	9091;
	xMsg9091.AmmInAdr	:=  iAdrAmmBase2MM;
	xMsg9091.AmmOutAdr	:=  iAdrMM2AmmBase;

	xMsg9096.Num		:=	9096;
	xMsg9096.AmmInAdr	:=  iAdrAmmBase2MM;
	xMsg9096.AmmOutAdr	:=  iAdrMM2AmmBase;

	xMsg9097.Num		:=	9097;
	xMsg9097.AmmInAdr	:=  iAdrAmmBase2MM;
	xMsg9097.AmmOutAdr	:=  iAdrMM2AmmBase;

	xMsg9214.Num		:=  9214;//SWAT920/5
	xMsg9214.AmmInAdr	:=  iAdrAmmBase2MM;
	xMsg9214.AmmOutAdr	:=  iAdrMM2AmmBase;

	xMsg9220.Num		:=  9220;//SWAT920/5a
	xMsg9220.AmmInAdr	:=  iAdrAmmBase2MM;
	xMsg9220.AmmOutAdr	:=  iAdrMM2AmmBase;

	xMsg9221.Num		:=	9221;
	xMsg9221.AmmInAdr	:=  iAdrAmmBase2MM;
	xMsg9221.AmmOutAdr	:=  iAdrMM2AmmBase;

	xMsg9222.Num		:=	9222;
	xMsg9222.AmmInAdr	:=  iAdrAmmBase2MM;
	xMsg9222.AmmOutAdr	:=  iAdrMM2AmmBase;

	xMsg9224.Num		:=	9224;
	xMsg9224.AmmInAdr	:=  iAdrAmmBase2MM;
	xMsg9224.AmmOutAdr	:=  iAdrMM2AmmBase;

	xMsg9225.Num		:=	9225;
	xMsg9225.AmmInAdr	:=  iAdrAmmBase2MM;
	xMsg9225.AmmOutAdr	:=  iAdrMM2AmmBase;

	xMsg9227.Num		:=	9227;
	xMsg9227.AmmInAdr	:=  iAdrAmmBase2MM;
	xMsg9227.AmmOutAdr	:=  iAdrMM2AmmBase;

	xMsg9254.Num		:=	9254;
	xMsg9254.AmmInAdr	:=  iAdrAmmBase2MM;
	xMsg9254.AmmOutAdr	:=  iAdrMM2AmmBase;

	xMsg9255.Num		:=	9255;
	xMsg9255.AmmInAdr	:=  iAdrAmmBase2MM;
	xMsg9255.AmmOutAdr	:=  iAdrMM2AmmBase;

	xMsg9256.Num		:=	9256;
	xMsg9256.AmmInAdr	:=  iAdrAmmBase2MM;
	xMsg9256.AmmOutAdr	:=  iAdrMM2AmmBase;

	xMsg9257.Num		:=	9257;
	xMsg9257.AmmInAdr	:=  iAdrAmmBase2MM;
	xMsg9257.AmmOutAdr	:=  iAdrMM2AmmBase;

	xMsg9258.Num		:=	9258;
	xMsg9258.AmmInAdr	:=  iAdrAmmBase2MM;
	xMsg9258.AmmOutAdr	:=  iAdrMM2AmmBase;

	xMsg9279.Num		:=	9279;
	xMsg9279.AmmInAdr	:=  iAdrAmmBase2MM;
	xMsg9279.AmmOutAdr	:=  iAdrMM2AmmBase;

	xMsg9280.Num		:=	9280;
	xMsg9280.AmmInAdr	:=  iAdrAmmBase2MM;
	xMsg9280.AmmOutAdr	:=  iAdrMM2AmmBase;

	xMsg9281.Num		:=	9281;
	xMsg9281.AmmInAdr	:=  iAdrAmmBase2MM;
	xMsg9281.AmmOutAdr	:=  iAdrMM2AmmBase;

	xMsg9282.Num		:=	9282;
	xMsg9282.AmmInAdr	:=  iAdrAmmBase2MM;
	xMsg9282.AmmOutAdr	:=  iAdrMM2AmmBase;

	xMsg9283.Num		:=	9283;
	xMsg9283.AmmInAdr	:=  iAdrAmmBase2MM;
	xMsg9283.AmmOutAdr	:=  iAdrMM2AmmBase;

	xMsg9303.Num		:=	9303;
	xMsg9303.AmmInAdr	:=  iAdrAmmBase2MM;
	xMsg9303.AmmOutAdr	:=  iAdrMM2AmmBase;

	xMsg9314.Num		:=	9314;
	xMsg9314.AmmInAdr	:=  iAdrAmmBase2MM;
	xMsg9314.AmmOutAdr	:=  iAdrMM2AmmBase;

	xMsg9316.Num		:=	9316;
	xMsg9316.AmmInAdr	:=  iAdrAmmBase2MM;
	xMsg9316.AmmOutAdr	:=  iAdrMM2AmmBase;

	xMsg9317.Num		:=	9317;
	xMsg9317.AmmInAdr	:=  iAdrAmmBase2MM;
	xMsg9317.AmmOutAdr	:=  iAdrMM2AmmBase;

	xMsg9322.Num		:=	9322;
	xMsg9322.AmmInAdr	:=  iAdrAmmBase2MM;
	xMsg9322.AmmOutAdr	:=  iAdrMM2AmmBase;

	xMsg9323.Num		:=	9323;
	xMsg9323.AmmInAdr	:=  iAdrAmmBase2MM;
	xMsg9323.AmmOutAdr	:=  iAdrMM2AmmBase;

	xMsg9324.Num		:=	9324;
	xMsg9324.AmmInAdr	:=  iAdrAmmBase2MM;
	xMsg9324.AmmOutAdr	:=  iAdrMM2AmmBase;

	xMsg9325.Num		:=	9325;
	xMsg9325.AmmInAdr	:=  iAdrAmmBase2MM;
	xMsg9325.AmmOutAdr	:=  iAdrMM2AmmBase;

	xMsg9326.Num		:=	9326;
	xMsg9326.AmmInAdr	:=  iAdrAmmBase2MM;
	xMsg9326.AmmOutAdr	:=  iAdrMM2AmmBase;

	xMsg9327.Num		:=	9327;
	xMsg9327.AmmInAdr	:=  iAdrAmmBase2MM;
	xMsg9327.AmmOutAdr	:=  iAdrMM2AmmBase;

	xMsg9328.Num		:=	9328;
	xMsg9328.AmmInAdr	:=  iAdrAmmBase2MM;
	xMsg9328.AmmOutAdr	:=  iAdrMM2AmmBase;

	xMsg9332.Num		:=	9332;
	xMsg9332.AmmInAdr	:=  iAdrAmmBase2MM;
	xMsg9332.AmmOutAdr	:=  iAdrMM2AmmBase;

	xMsg9333.Num		:=	9333;
	xMsg9333.AmmInAdr	:=  iAdrAmmBase2MM;
	xMsg9333.AmmOutAdr	:=  iAdrMM2AmmBase;

	xMsg9334.Num		:=	9334;
	xMsg9334.AmmInAdr	:=  iAdrAmmBase2MM;
	xMsg9334.AmmOutAdr	:=  iAdrMM2AmmBase;

	xMsg9335.Num		:=	9335;
	xMsg9335.AmmInAdr	:=  iAdrAmmBase2MM;
	xMsg9335.AmmOutAdr	:=  iAdrMM2AmmBase;

	xMsg9336.Num		:=	9336;
	xMsg9336.AmmInAdr	:=  iAdrAmmBase2MM;
	xMsg9336.AmmOutAdr	:=  iAdrMM2AmmBase;

	xMsg9352.Num		:=	9352;
	xMsg9352.AmmInAdr	:=  iAdrAmmBase2MM;
	xMsg9352.AmmOutAdr	:=  iAdrMM2AmmBase;

	xMsg9353.Num		:=	9353;
	xMsg9353.AmmInAdr	:=  iAdrAmmBase2MM;
	xMsg9353.AmmOutAdr	:=  iAdrMM2AmmBase;

	xMsg9354.Num		:=	9354;
	xMsg9354.AmmInAdr	:=  iAdrAmmBase2MM;
	xMsg9354.AmmOutAdr	:=  iAdrMM2AmmBase;

	xMsg9355.Num		:=	9355;
	xMsg9355.AmmInAdr	:=  iAdrAmmBase2MM;
	xMsg9355.AmmOutAdr	:=  iAdrMM2AmmBase;

	xMsg9356.Num		:=	9356;
	xMsg9356.AmmInAdr	:=  iAdrAmmBase2MM;
	xMsg9356.AmmOutAdr	:=  iAdrMM2AmmBase;

	xMsg9357.Num		:=	9357;
	xMsg9357.AmmInAdr	:=  iAdrAmmBase2MM;
	xMsg9357.AmmOutAdr	:=  iAdrMM2AmmBase;

	xMsg9358.Num		:=	9358;
	xMsg9358.AmmInAdr	:=  iAdrAmmBase2MM;
	xMsg9358.AmmOutAdr	:=  iAdrMM2AmmBase;

	xMsg9359.Num		:=	9359;
	xMsg9359.AmmInAdr	:=  iAdrAmmBase2MM;
	xMsg9359.AmmOutAdr	:=  iAdrMM2AmmBase;

	xMsg9362.Num		:=	9362;			(*V4.12 Oil Tank*)
	xMsg9362.AmmInAdr	:=  iAdrAmmBase2MM;
	xMsg9362.AmmOutAdr	:=  iAdrMM2AmmBase;

	xMsg9363.Num		:=	9363;			(*V4.12 Oil Tank*)
	xMsg9363.AmmInAdr	:=  iAdrAmmBase2MM;
	xMsg9363.AmmOutAdr	:=  iAdrMM2AmmBase;

	xMsg9364.Num		:=	9364;			(*V4.12 Oil Tank*)
	xMsg9364.AmmInAdr	:=  iAdrAmmBase2MM;
	xMsg9364.AmmOutAdr	:=  iAdrMM2AmmBase;

	xMsg9369.Num		:=	9369;
	xMsg9369.AmmInAdr	:=  iAdrAmmBase2MM;
	xMsg9369.AmmOutAdr	:=  iAdrMM2AmmBase;

	xMsg9378.Num		:=	9378;
	xMsg9378.AmmInAdr	:=  iAdrAmmBase2MM;
	xMsg9378.AmmOutAdr	:=  iAdrMM2AmmBase;

	xMsg9390.Num		:=	9390;
	xMsg9390.AmmInAdr	:=  iAdrAmmBase2MM;
	xMsg9390.AmmOutAdr	:=  iAdrMM2AmmBase;

	xMsg9435.Num		:=  9435;
	xMsg9435.AmmInAdr	:=  iAdrAmmBase2MM;
	xMsg9435.AmmOutAdr	:=  iAdrMM2AmmBase;

	xMsg9436.Num		:=  9436;
	xMsg9436.AmmInAdr	:=  iAdrAmmBase2MM;
	xMsg9436.AmmOutAdr	:=  iAdrMM2AmmBase;

	xMsg9513.Num		:=	9513;
	xMsg9513.AmmInAdr	:=  iAdrAmmBase2MM;
	xMsg9513.AmmOutAdr	:=  iAdrMM2AmmBase;

	xMsg9560.Num		:=  9560;
	xMsg9560.AmmInAdr	:=  iAdrAmmBase2MM;
	xMsg9560.AmmOutAdr	:=  iAdrMM2AmmBase;

	xMsg9561.Num		:=  9561;
	xMsg9561.AmmInAdr	:=  iAdrAmmBase2MM;
	xMsg9561.AmmOutAdr	:=  iAdrMM2AmmBase;

	(* template
	xMsg.Num		:=	;
	xMsg.AmmInAdr	:=  iAdrAmmBase2MM;
	xMsg.AmmOutAdr	:=  iAdrMM2AmmBase;
	*)
END_PROGRAM
```

#### MsgAG.var
```iecst
VAR
	bAnyHWC_SL_FailActive : BOOL;
	bHWC_SL_Active : BOOL;
	HBT_3 : BOOL; (*Failure motor cooling water pump*)
	HBT_4 : BOOL;
	HBT_5 : BOOL;
	HBT_6 : BOOL;
	HBT_7 : BOOL;
	HBT_8 : BOOL;
	iAdrAmmBase2MM : UDINT;
	iAdrMM2AmmBase : UDINT;
	xGR_MAXR_1120 : GR_MAXR;
	xTOF_CCWP_Fail : TOF;
	xTOF_ECWP_PreH_FS : TOF;
	xTOF_EngAuxMon : TOF;
	xTOF_EngDemEPS : TOF;
	xTOF_HWP_Fail : TOF;
	xTON_1120 : TON;
	xTON_ECWP_PreH_Mon : TON;
	xTON_HWP_Fail : TON;
	xTON_PrGO_Lo : TON;
	xTON_PrGO_Rel : TON;
	xGR_MIN_Pr_TCO_Lo : GR_MINR;
	xGR_MAXR_Pr_TCO_hihi : GR_MAXR;
	xTON_Pr_TCO_Mon : TON;
	xGR_MAXR_Pr_TCO_hi : GR_MAXR;
	xGR_MAXR_OTMAA : GR_MAXR;
	xGR_MAXR_OTMA : GR_MAXR;
	xGR_MAXR_OTMA_Prio2 : GR_MAXR;
	xTON_BRTB_60s : TON;
	xTON_OTMAA : TON;
	xTON_OTMA : TON;
	xTON_OT : TON;
	xTON_OT_Prio2 : TON;
	AN_OTMA : BOOL; (* Öltemperatur maximum *)
	AN_OTMA_Prio2 : BOOL; (* Oil temperature maximum Prio2*)
	AN_OTMAA : BOOL; (* Öltemperatur max Sofortabstellung *)
	T_OTMA : BOOL; (* Öltemperatur maximum *)
	M_OMIN_DREHZ : BOOL;
	xTON_OilPreH_Of : TON;
	xTON_OilPreH_On : TON;
	xF_TRIG_ACP_Start : F_TRIG;
	xMsg1017 : Msg;
	xMsg1018 : Msg;
	xMsg1020 : Msg;
	xMsg1023 : Msg;
	xMsg1043 : Msg;
	xMsg1051 : Msg;
	xMsg1052 : Msg;
	xMsg1053 : Msg;
	xMsg1054 : Msg;
	xMsg1059 : Msg;
	xMsg1060 : Msg;
	xMsg1090 : Msg;
	xMsg1091 : Msg;
	xMsg1100 : Msg;
	xMsg1101 : Msg;
	xMsg1120 : Msg;
	xMsg1129 : Msg;
	xMsg1137 : Msg;
	xMsg1139 : Msg;
	xMsg1140 : Msg;
	xMsg1148 : Msg;
	xMsg1159 : Msg;
	xMsg1160 : Msg;
	xMsg1166 : Msg;
	xMsg1249 : Msg;
	xMsg1250 : Msg;
	xMsg1257 : Msg;
	xMsg1258 : Msg;
	xMsg1259 : Msg;
	xMsg1260 : Msg;
	xMsg1261 : Msg;
	xMsg1262 : Msg;
	xMsg1263 : Msg;
	xMsg1264 : Msg;
	xMsg1281 : Msg;
	xMsg1282 : Msg;
	xMsg1292 : Msg; (*Manual operating auxiliaries control - Handbedienebene*)
	xMsg2102 : Msg;
	xMsg2103 : Msg;
	xMsg2114 : Msg;
	xMsg2118 : Msg;
	xMsg2201 : Msg;
	xMsg2213 : Msg;
	xMsg2224 : Msg;
	xMsg2233 : Msg;
	xMsg2234 : Msg;
	xMsg2238 : Msg;
	xMsg2242 : Msg;
	xMsg2260 : Msg;
	xMsg2263 : Msg;
	xMsg2264 : Msg;
	xMsg2265 : Msg;
	xMsg2266 : Msg;
	xMsg2267 : Msg;
	xMsg2268 : Msg;
	xMsg2269 : Msg;
	xMsg2284 : Msg;
	xMsg2291 : Msg;
	xMsg2292 : Msg;
	xMsg2304 : Msg;
	xMsg2332 : Msg;
	xMsg2333 : Msg;
	xMsg2348 : Msg;
	xMsg2349 : Msg;
	xMsg2350 : Msg;
	xMsg2351 : Msg;
	xMsg2352 : Msg;
	xMsg2353 : Msg;
	xMsg2355 : Msg;
	xMsg2359 : Msg;
	xMsg2360 : Msg;
	xMsg2361 : Msg;
	xMsg2376 : Msg; (*Scavenging by starting system not successful*)
	xMsg2377 : Msg; (*Measuring signal failure voltage start motor 1 *)
	xMsg2378 : Msg; (*Measuring signal failure voltage start motor 1 *)
	xMsg2379 : Msg; (*Measuring signal failure voltage start motor 1 *)
	xMsg2382 : Msg; (*Start attempt failed minimum speed*)
	xMsg2421 : Msg;
	xMsg2422 : Msg;
	xMsg2423 : Msg; (*SWAT920/1*)
	xMsg2424 : Msg; (*SWAT920/2*)
	xMsg2425 : Msg; (*SWAT920/2*)
	xMsg2426 : Msg; (*SWAT920/2*)
	xMsg2427 : Msg;
	xMsg2431 : Msg; (*SWAT920/1*)
	xMsg2432 : Msg; (*SWAT920/1*)
	xMsg2433 : Msg; (*SWAT920/1*)
	xMsg2434 : Msg;
	xMsg2435 : Msg; (*SWAT920/2*)
	xMsg2459 : Msg;
	xMsg2473 : Msg;
	xMsg2475 : Msg;
	xMsg2524 : Msg;
	xMsg2534 : Msg;
	xMsg2545 : Msg;
	xMsg2554 : Msg;
	xMsg2557 : Msg; (*SWAT920/2*)
	xMsg2558 : Msg;
	xMsg2559 : Msg;
	xMsg2560 : Msg;
	xMsg2571 : Msg;
	xMsg2572 : Msg;
	xMsg2576 : Msg;
	xMsg2579 : Msg;
	xMsg2582 : Msg;
	xMsg2587 : Msg;
	xMsg2589 : Msg;
	xMsg2590 : Msg;
	xMsg2591 : Msg;
	xMsg2592 : Msg;
	xMsg2594 : Msg;
	xMsg2595 : Msg;
	xMsg2596 : Msg;
	xMsg2597 : Msg;
	xMsg2598 : Msg;
	xMsg2599 : Msg;
	xMsg2600 : Msg;
	xMsg2602 : Msg;
	xMsg2603 : Msg;
	xMsg2604 : Msg;
	xMsg2605 : Msg;
	xMsg2606 : Msg;
	xMsg2608 : Msg;
	xMsg2613 : Msg;
	xMsg2624 : Msg;
	xMsg2625 : Msg;
	xMsg2627 : Msg;
	xMsg2628 : Msg;
	xMsg2629 : Msg;
	xMsg2636 : Msg;
	xMsg2642 : Msg;
	xMsg2643 : Msg;
	xMsg2644 : Msg;
	xMsg2645 : Msg;
	xMsg2646 : Msg;
	xMsg2648 : Msg;
	xMsg2649 : Msg; (*W2649 Crank case pressure low  *)
	xMsg2650 : Msg; (*W2650 Blow by blower not ready  *)
	xMsg2651 : Msg; (*W2651 Measuring signal failure pressure before blow by filter  *)
	xMsg2652 : Msg; (*W2652 Measuring signal failure pressure after blow by filter  *)
	xMsg2653 : Msg; (*W2653 Blow by filter difference pressure high - maintenance  *)
	xMsg2654 : Msg; (*W2654 Blow by filter difference pressure low  *)
	xMsg2666 : Msg;
	xMsg2689 : Msg;
	xMsg2722 : Msg;
	xMsg2723 : Msg;
	xMsg2724 : Msg;
	xMsg2725 : Msg;
	xMsg2726 : Msg;
	xMsg2727 : Msg;
	xMsg2728 : Msg;
	xMsg2729 : Msg;
	xMsg2737 : Msg;
	xMsg2738 : Msg;
	xMsg2739 : Msg;
	xMsg2740 : Msg;
	xMsg2741 : Msg;
	xMsg2742 : Msg;
	xMsg2754 : Msg;
	xMsg2755 : Msg;
	xMsg2756 : Msg;
	xMsg2757 : Msg;
	xMsg2758 : Msg;
	xMsg2759 : Msg;
	xMsg2760 : Msg;
	xMsg2761 : Msg;
	xMsg2762 : Msg;
	xMsg2770 : Msg;
	xMsg2771 : Msg;
	xMsg2772 : Msg;
	xMsg2773 : Msg;
	xMsg2774 : Msg;
	xMsg2775 : Msg;
	xMsg2776 : Msg;
	xMsg2777 : Msg;
	xMsg2778 : Msg;
	xMsg2781 : Msg;
	xMsg2782 : Msg;
	xMsg2783 : Msg;
	xMsg2784 : Msg;
	xMsg2785 : Msg;
	xMsg2786 : Msg;
	xMsg2787 : Msg;
	xMsg2788 : Msg;
	xMsg2789 : Msg;
	xMsg2791 : Msg;
	xMsg2792 : Msg;
	xMsg2809 : Msg;
	xMsg2810 : Msg;
	xMsg2931 : Msg;
	xMsg2932 : Msg;
	xMsg2933 : Msg;
	xMsg2956 : Msg;
	xMsg2957 : Msg;
	xMsg2978 : Msg;
	xMsg2979 : Msg;
	xMsg3216 : Msg;
	xMsg3218 : Msg;
	xMsg3300 : Msg;
	xMsg3301 : Msg;
	xMsg3304 : Msg;
	xMsg3305 : Msg;
	xMsg3322 : Msg;
	xMsg3323 : Msg;
	xMsg3350 : Msg;
	xMsg3351 : Msg;
	xMsg3369 : Msg;
	xMsg3370 : Msg;
	xMsg3375 : Msg;
	xMsg3401 : Msg;
	xMsg3403 : Msg;
	xMsg3405 : Msg;
	xMsg3413 : Msg;
	xMsg3414 : Msg;
	xMsg3415 : Msg;
	xMsg3416 : Msg;
	xMsg3495 : Msg;
	xMsg3496 : Msg;
	xMsg3497 : Msg;
	xMsg3507 : Msg;
	xMsg3515 : Msg;
	xMsg3519 : Msg;
	xMsg3572 : Msg;
	xMsg3574 : Msg;
	xMsg3578 : Msg;
	xMsg3579 : Msg;
	xMsg3587 : Msg;
	xMsg3588 : Msg;
	xMsg9214 : Msg; (*SWAT920/5*)
	xMsg9220 : Msg; (*SWAT920/5a*)
	xMsg9221 : Msg;
	xMsg9222 : Msg;
	xMsg9224 : Msg;
	xMsg9225 : Msg;
	xMsg9227 : Msg;
	xMsg9254 : Msg;
	xMsg9255 : Msg;
	xMsg9256 : Msg;
	xMsg9257 : Msg;
	xMsg9258 : Msg;
	xMsg9279 : Msg;
	xMsg9280 : Msg;
	xMsg9281 : Msg;
	xMsg9282 : Msg;
	xMsg9283 : Msg;
	xMsg9303 : Msg;
	xMsg9314 : Msg;
	xMsg9316 : Msg;
	xMsg9317 : Msg;
	xMsg9001 : Msg;
	xMsg9002 : Msg;
	xMsg9003 : Msg;
	xMsg9048 : Msg;
	xMsg9067 : Msg;
	xMsg9069 : Msg;
	xMsg9070 : Msg;
	xMsg9074 : Msg;
	xMsg9088 : Msg; (*Scavenging by starting system successful*)
	xMsg9089 : Msg; (*Starter motor 1 did not engage*)
	xMsg9090 : Msg; (*Starter motor 2 did not engage*)
	xMsg9091 : Msg; (*Starter motor 3 did not engage*)
	xMsg9096 : Msg; (*Starter overheated*)
	xMsg9097 : Msg; (*Purge cranking cycle initiated*)
	xMsg9322 : Msg;
	xMsg9323 : Msg;
	xMsg9324 : Msg;
	xMsg9325 : Msg;
	xMsg9326 : Msg;
	xMsg9327 : Msg;
	xMsg9328 : Msg;
	xMsg9332 : Msg;
	xMsg9333 : Msg;
	xMsg9334 : Msg;
	xMsg9335 : Msg;
	xMsg9336 : Msg;
	xMsg9352 : Msg;
	xMsg9353 : Msg;
	xMsg9354 : Msg;
	xMsg9355 : Msg;
	xMsg9356 : Msg;
	xMsg9357 : Msg;
	xMsg9358 : Msg;
	xMsg9359 : Msg;
	xMsg9369 : Msg;
	xMsg9378 : Msg; (*V4.13*)
	xMsg9390 : Msg; (*Oil temperature before engine start too low*)
	xMsg9435 : Msg; (*FuB*) (*SAFETY PLC*)
	xMsg9436 : Msg; (*FuB*) (*SAFETY PLC*)
	xMsg9513 : Msg; (*Failure engine oil refilling*) (*2024-225*)
	xMsg9560 : Msg; (*FuB*) (*SAFETY PLC*)
	xMsg9561 : Msg; (*FuB*) (*SAFETY PLC*)
	TON_FOP : TON;
	bFOP_LZ_max : BOOL;
	xR_TRIG_N_TCO_FS : R_TRIG;
	GR_MIN_OIL_STARTFG : GR_MINR;
	xTOF_CC2WP_Fail : TOF;
	bPLC_Startup : BOOL;
	xTOF_EmCWP_Fail : TOF;
	xTON_EmCWP_Dem : TON;
	iIdx_CtrlBat : USINT;
	bAMM_CtrlBat_ChargeDev_Fail : BOOL;
	xMsg9362 : Msg; (*V4.12*)
	xMsg9363 : Msg; (*V4.12*)
	xMsg9364 : Msg; (*V4.12*)
	rDPr_ECWP1 : REAL; (*cooling water difference pressure over ECWP1 (M.04-PI-010 minus M.04-PI-001)*)
	rDPr_ECWP2 : REAL; (*cooling water difference pressure over ECWP2 (M.04-PI-011 minus M.04-PI-001)*)
	xTON_DPr_ECWP_MonRel : TON;
	xTON_DPr_ECWP_LoLo : TON;
	xTON_EleStarter_Dem : TON; (*Starter MSF detection delay*)
	xRT_EleStarter_Dem : R_TRIG; (*Starter MSF detection trigger*)
	xTON_Msg9222 : TON; (*FuB*)
	xTON_Msg9225 : TON; (*FuB*)
END_VAR
```

### Program Logical/AuxiliariesGeneral/Vis_AG (IEC, version 4.14.0) - visualization

#### Vis_AGCyclic.st
```iecst
(*******************************************************************************
vis			visualization

This code is confidential and proprietary to the INNIO Company.
It may not be used in any form, or reproduced in any manner,
without the express written permission of the INNIO Company.
Copyright, INNIO Company, 2024

Customized modifications: -
------------------------

History:
-------
V0.00.0	24.04.2012	lettenb.	new
V3.99.0	25.04.2013	lettenb.	data for oil counter trending added
		03.05.2013				ctr input var's from vis moved to Ctr_EO
		16.05.2013				MM2VIS.rOC_Consum_Avg added
V3.99.1	21.08.2013	Denk		Oil quality sensor added
V4.00.0	30.06.2014	lettenb.	MM2VIS.bECWP1Dem: xEngType.Type2 added, bugfix
		20.11.2014				920: engine bearing removed --> MM_EG
		26.01.2015				920: Ctr_EOVal_LT, Ctr_EOVal_LT added
V4.03.0 07.08.2015  Denk		Manual operating auxiliaries control functionality added
		11.01.2016				MM2VIS oil counter interfaces moved from Vis_AG -> Cnt_EO(to enable scroll function of settings)bugfix
V4.04.0	10.05.2016	lettenb.	rPr_EOaP added
V4.05.0	10.05.2016	lettenb.	prelubrication for fast start
V4.05.1	19.02.2018	lettenb.	rDPr_BbFilt_A,rDPr_BbFilt_B prepared for vis
V4.06.0	19.09.2018	Perktold, 	integrated MM2VIS.bPreL_FS_EngStaRel
V4.07.0	17.12.2018	Schmid		hydraulic ECW pre-heating added
		08.01.2019	Schmid		redundant pump control
V4.09.0	11.12.2019	Schmid		new air starter design: engagement pressure sensor and valve commands added
V4.10.0	12.01.2020	Schmid		added MM2VIS.bNoExtendedPrelube for 5min start
		16.12.2020	Schmid		battery voltages added
V4.11.0	05.11.2021	Schmid		added OUT_AG.bECWP_MechDriven for Pr_ECW plausibility check
V4.12.0	06.12.2022 	Bacci		control cabinet battery voltages bugfixing
		24.02.2023	Tinello		added MM2VIS for HWP
V4.13.0	27.09.2023	Bacci		MM2VIS.rOQS_Temp, MM2VIS.rOQS_Visco, MM2VIS.rOQS_Dielect, MM2VIS.rOQS_Conduct deleted
		01.02.2024	Tinello		Only one calculation for oil filter diff pressure (2023-184)
		15.02.2024	Bacci		MM2VIS.bU_Starter_engage1 added
V4.14.0	25.11.2024  Bacci		T6 Start procedure with purge start (2024-219): added volume of purge air, purge state, fast start readiness

Instructions for use:
--------------------
Outstandings:
------------
*******************************************************************************)
PROGRAM _CYCLIC

	MM2VIS.rPr_CC      				:= IN_AG.tPr_CC.Ai;

	MM2VIS.bEOP1AC_Dem 				:= OUT_AG.tEOP1AC_Dem.Do;
	MM2VIS.bEOP1DC_Dem 				:= OUT_AG.tEOP1DC_Dem.Do;

	IF Para.bECWP_MechDriven AND (xEngType.Type2 OR xEngType.Type3) THEN
		MM2VIS.bECWP1Dem			:=	M_DREHZ;
		OUT_AG.bECWP_MechDriven		:=	TRUE;		(*custom new Pr_ECW plausibility check*)
	ELSE
		MM2VIS.bECWP1Dem			:=	OUT_AG.tECWP1Dem.Do;
		OUT_AG.bECWP_MechDriven		:=	FALSE;		(*custom new Pr_ECW plausibility check*)
	END_IF;

	MM2VIS.bECWP2Dem      			:= OUT_AG.tECWP2Dem.Do;
	MM2VIS.bECWP_PreH_Dem 			:= OUT_AG.tECWP_PreH_Dem.Do;
	MM2VIS.bECW_PreH_Dem  			:= OUT_AG.tECW_PreH_Dem.Do;
	MM2VIS.bECW_PreHV_Opened  		:= IN_AG.tECW_PreHV_Opened.Di;
	MM2VIS.bECW_CV_Open		    	:= bECW_CV_Open;
	MM2VIS.rCtr_ECW_Set				:= OUT_AG.tCtr_ECW_Set.Ao;
	MM2VIS.rPr_ECWaP1				:= IN_AG.tPr_ECWaP1.Ai;
	MM2VIS.rPr_ECWaP2				:= IN_AG.tPr_ECWaP2.Ai;

	MM2VIS.bPreL_FS_EngStaRel		:= OUT_AG.bPreL_FS_EngStaRel AND OUT_AG.bT_EOP_RelFS AND (Para.bFSPreL_Act OR xEngType.Type3);
	MM2VIS.bNoExtendedPrelube		:= OUT_AG.bNoExtendedPrelube;

	MM2VIS.bEng_StaSpdExc			:= M_DREHZ;
	MM2VIS.rPr_EOF_Diff				:= rDPr_EOF;

	MM2VIS.rPr_EngLubOil 			:= IN_AG.tPr_EngLubOil.Ai;
	MM2VIS.rPr_EOF_DiffMon 			:= IN_AG.tPr_EOF_DiffMon.Ai;	(* engine oil pressure before filter *)
	MM2VIS.rEO_Level 				:= IN_AG.tEO_Level.Ai;
	MM2VIS.rPr_EOF_After			:= IN_AG.tPr_EOF_After.Ai;
	MM2VIS.rPr_EOaP					:= IN_AG.tPr_EOaP.Ai;			(* engine oil pressure after pump *)
	MM2VIS.rT_EO					:= IN_AG.tT_EO.Ai;
	MM2VIS.rT_EOP_After				:= IN_AG.tT_EOP_After.Ai;

	MM2VIS.rPr_TC_EOF_After			:= IN_AG.tPr_TC_EOF_After.Ai;
	MM2VIS.rPr_TC_EOF_Before		:= IN_AG.tPr_TC_EOF_Before.Ai;
	MM2VIS.rPr_Oil_LPTC_In_A		:= IN_AG.tPr_Oil_LPTC_In_A.Ai;
	MM2VIS.rPr_Oil_LPTC_In_B		:= IN_AG.tPr_Oil_LPTC_In_B.Ai;
	MM2VIS.rPr_TCO		 			:= IN_AG.tPr_TCO.Ai;
	MM2VIS.bTCOV_CoClose 			:= OUT_AG.tTCOV_CoClose.Do;

	MM2VIS.rT_EO_Pan				:= IN_AG.tT_EO_Pan.Ai;
	MM2VIS.rT_EO_Preheating			:= IN_AG.tT_EO_Preheating.Ai;
	MM2VIS.bEOF_PreheatRel			:= OUT_AG.tEOF_PreheatRel.Do;
	MM2VIS.bEO_Preheat1				:= OUT_AG.tEO_Preheat1.Do;
	MM2VIS.bEO_Preheat2				:= OUT_AG.tEO_Preheat2.Do;
	MM2VIS.bEO_Preheat3				:= OUT_AG.tEO_Preheat3.Do;

	(*BlowBy*)
	MM2VIS.rPr_f_BbFilt				:= IN_AG.tPr_f_BbFilt.Ai;
	MM2VIS.rPr_a_BbFilt				:= IN_AG.tPr_a_BbFilt.Ai;
	MM2VIS.rPr_f_BbFilt_A			:= IN_AG.tPr_f_BbFilt_A.Ai;
	MM2VIS.rPr_a_BbFilt_A			:= IN_AG.tPr_a_BbFilt_A.Ai;
	MM2VIS.rPr_f_BbFilt_B			:= IN_AG.tPr_f_BbFilt_B.Ai;
	MM2VIS.rPr_a_BbFilt_B			:= IN_AG.tPr_a_BbFilt_B.Ai;
	MM2VIS.rDPr_BbFilt				:= rDPr_BbFilt;
	MM2VIS.rDPr_BbFilt_A			:= rDPr_BbFilt_A;
	MM2VIS.rDPr_BbFilt_B			:= rDPr_BbFilt_B;

	(*EleStart*)
	MM2VIS.bU_Starter_engage1		:= IN_AG.tU_Starter_engage1.GoodQual;
	MM2VIS.iVol_PurgeAir			:= iVol_PurgeAir;
	MM2VIS.bSt_Purge				:= bSt_Purge;
	MM2VIS.bFS_Rdy_STT_StPurge		:= OUT_AG.bFS_Rdy_STT_StPurge OR NOT xEngType.Type6;
	MM2VIS.iTi_ST_Res				:= iTi_ST_Res;

	(*AirStart*)
	MM2VIS.rPr_AirStarter_Tank		:= IN_AG.tPr_AirStarter_Tank.Ai;
	MM2VIS.rPr_AirStarter_Supply	:= IN_AG.tPr_AirStarter_Supply.Ai;
	MM2VIS.rN_AirStarter			:= rN_AirStarter;
	MM2VIS.rPr_AirST_Engage			:= IN_AG.tPr_AirST_Engage.Ai;
	MM2VIS.bAirST_ValEngage			:= OUT_AG.tAirST_ValEngage.Do;
	MM2VIS.bAirST_ValStart			:= OUT_AG.tAirST_ValStart.Do;

	(* Manual operating auxiliaries control - Handbedienebene *)
	MM2VIS.bManOpAuxCtr_Gnl_Rel		:= OUT_AG.tManAuxCtr.bGnl_Rel;		(* General release for button MAN/AUTO visibility *)

	(* Hydraulic ECW pre-heating *)
	MM2VIS.bECW_HydrPreH_Dem		:= bECW_HydrPreH_Dem;
	MM2VIS.rT_HW_Su_PreH_ECW_LimLo	:= IN_AG.tT_ECW.Ai + 10.0;
	MM2VIS.rT_HW_Su_PreH_ECW_LimHi	:= 95.0;

	(* Heating water pump *)
	MM2VIS.bHWP_On					:= OUT_AG.tHWP_Dem.Do 		AND IN_AG.tHWP_Op.Di;

	(* Redundant heating water pumps *)
	MM2VIS.bHWP1_Op					:= OUT_AG.tHWP1_Dem.Do		AND IN_AG.tHWP1_Op.Di;
	MM2VIS.bHWP2_Op					:= OUT_AG.tHWP2_Dem.Do		AND IN_AG.tHWP2_Op.Di;
	(* Redundant charge cooler water pumps *)
	MM2VIS.bCCWP1_Op				:= OUT_AG.tCCWP1_Dem.Do		AND IN_AG.tCCWP1_Op.Di;
	MM2VIS.bCCWP2_Op				:= OUT_AG.tCCWP2_Dem.Do		AND IN_AG.tCCWP2_Op.Di;
	(* Redundant charge cooler 2 water pumps *)
	MM2VIS.bCC2WP1_Op				:= OUT_AG.tCC2WP1_Dem.Do	AND IN_AG.tCC2WP1_Op.Di;
	MM2VIS.bCC2WP2_Op				:= OUT_AG.tCC2WP2_Dem.Do	AND IN_AG.tCC2WP2_Op.Di;
	(* Redundant emergency cooler water pumps *)
	MM2VIS.bEmCWP1_Op				:= OUT_AG.tEmCWP1_Dem.Do	AND IN_AG.tEmCWP1_Op.Di;
	MM2VIS.bEmCWP2_Op				:= OUT_AG.tEmCWP2_Dem.Do	AND IN_AG.tEmCWP2_Op.Di;

	(* Battery voltages *)
	MM2VIS.rU_StarterBat := IN_AG.tU_StarterBat.Ai;
	MM2VIS.rU_BufferBat1 := IN_AG.tU_BufferBat1.Ai;
	MM2VIS.rU_BufferBat2 := IN_AG.tU_BufferBat2.Ai;

	MM2VIS.bStarterBat_UnderTest   := bStarterBat_Disconnect;
	MM2VIS.bBufferBat_UnderTest[1] := OUT_AG.tBufferBat1_Disconnect.Do;
	MM2VIS.bBufferBat_UnderTest[2] := OUT_AG.tBufferBat2_Disconnect.Do;

	FOR iIdx_CtrlBat := 1 TO iNum_CtrlBatMon DO
		MM2VIS.rU_CtrlBat[iIdx_CtrlBat]				:=	IN_AG.tU_CtrlBat[iIdx_CtrlBat].Ai;
		MM2VIS.sLocIdent_CtrlBatMon[iIdx_CtrlBat]	:=	IN_AG.sLocIdent_CtrlBatMon[iIdx_CtrlBat];
		MM2VIS.bCtrlBat_UnderTest[iIdx_CtrlBat]     :=  OUT_AG.tCtrlBat_Disconnect[iIdx_CtrlBat].Do;
	END_FOR;

	MM2VIS.bCtrlBat_Used                            :=  bCtrlBat_Used;
	MM2VIS.iNumActive_CtrlBatMon					:=	iNr_CtrlBat_Used;

	MM2VIS.bU_StarterBat_Exist						:=	FALSE;

	(* Oil leakage affected additional oil tank - A2361 assistant value *)
	IF 		NOT IN_AG.tLeak_OilExtensionTank1.Di THEN	MM2VIS.iLeak_OilExtensionTank := 1;
	ELSIF	NOT IN_AG.tLeak_OilExtensionTank2.Di THEN	MM2VIS.iLeak_OilExtensionTank := 2;
	ELSIF	NOT IN_AG.tLeak_OilExtensionTank3.Di THEN	MM2VIS.iLeak_OilExtensionTank := 3;
	ELSE												MM2VIS.iLeak_OilExtensionTank := 0;
	END_IF;

END_PROGRAM
```

#### Vis_AG.var
```iecst
VAR
	iIdx_CtrlBat : USINT;
END_VAR
```

### Program Logical/AuxiliariesGeneral/ParAG (IEC, version 4.07.0) - + parameter handling

- perm_par.st (not readable text: treated as protected, skipped)

#### perm_par.var
```iecst
VAR
	tParaIntern : ParaHandler_typ; (*Connector type to perm_par*)
	tMM2ParaBase_ReadBack : MM2ParaBase_type; (*INTERNAL! V4.06 new readback structure for information from previous tasks*)
	bWriteDataObj : BOOL; (* TRUE=write data object module *)
	bDataObjLenErr : BOOL; (*Error occured in permem: data module size missmatch*)
	bCreateDataObj : BOOL; (* TRUE=create new data object *)
	bWriteOnce : BOOL; (* write permanent memory once *)
	DatObjCreate_01 : DatObjCreate; (* data object create *)
	DatObjInfoBak_02 : DatObjInfo; (* data object info *)
	DatObjDelete_01 : DatObjDelete; (* data object delete *)
	DatObjRead_01 : DatObjRead; (* data object read *)
	DatObjRead_02 : DatObjRead; (* manual initiated data object read *)
	DatObjWrite_01 : DatObjWrite; (* data object write *)
	DatObjDelete_02 : DatObjDelete; (* data object delete *)
	DatObjDelete_11 : DatObjDelete; (*Delete Backup File*)
	DatObjInfo_01 : DatObjInfo; (* data object info *)
	DatObjInfo_02 : DatObjInfo; (* data object info *)
	szModuleName : STRING[35]; (* module name of object *)
	szModuleNameBackup : STRING[35]; (* module name of posiibly created backup object *)
	DatObjCopy_01 : DatObjCopy;
	bCopyDataObj : BOOL;
	TON_WarnDelay : TON;
	TON_WritePMEM : TON; (* delay write permanent memory *)
	ulPMPointer : UDINT; (* adress of actual checksum value *)
	ulChecksum : UDINT; (* parameter checksum value *)
	pm_len : UDINT; (* permanent value lenght *)
	ulChecksumOld : UDINT; (* last vlaue of parameter checksum *)
	ulChkValue : UDINT; (* actual value of parameter pointer *)
	pm_id : UDINT; (* permanent value identifier *)
	pm_p : UDINT; (* permanent value pointer *)
	DatObjInfo_META : DatObjInfo;
	DatObjRead_META : DatObjRead;
	szMetaDataRaw : STRING[2000];
	szMetaData : ARRAY[0..4] OF STRING[35];
	szMetaDataVis : ARRAY[0..3] OF STRING[35];
	ssIndex : INT;
	ssCount : INT;
	ucMetaDataRaw : ARRAY[0..2000] OF USINT;
	ssCount2 : INT;
	szMetaDataFile : STRING[10];
	szText1 : STRING[20];
	pv_adr_IN_XX_tPB2MM : UDINT;
	pv_lng : UDINT;
	pv_lng_IN_XX_tPB2MM : UDINT;
	pv_lng_OUT_XX_tPB2MM : UDINT;
	szText2 : STRING[20];
	pv_adr_OUT_XX_tXX2PB : UDINT;
END_VAR
VAR CONSTANT
	ERR_NOERROR : UINT := 0;
END_VAR
VAR
	usPMWriteCnt : UINT;
	pm_Error : UDINT; (* permanent value error *) (* Deleted: pm : ParaMem_typ; permanent memory tags mathias, 22.8.11*)
	fun_Error : UDINT := 0; (*state > 0 = function error*)
	xLocalParaCheck : ParaCheckFUB; (*local function instance to check parameter values*)
	TON_ParaSetupOk : TON;
	bParaCheckSystemOk : BOOL;
	iDebug_ParaOkChecked : UDINT;
	bRestoreBackupDataObj : BOOL := FALSE;
	bRestoreDataObjContent : BOOL := FALSE;
	pm_id_backup : UDINT;
	pm_p_Backup : UDINT;
	DatObjCopy_02 : DatObjCopy;
	bDeleteBackupDataObj : BOOL := FALSE; (*Command to delete backup data module file on purpose*)
	bDebugPara : ARRAY[0..5] OF BOOL;
	ssIndex2 : INT;
	ssIndex3 : INT;
	ssIndex4 : INT;
	ssIndexVis : INT;
	szText : STRING[40];
	pv_adr_Para : UDINT;
	szParaSnippet : ARRAY[0..5] OF STRING[150];
	szParaIndex : STRING[10];
	slValue : DINT;
	iModuleDLD_ResetCount : INT;
	bDownloadDetected : BOOL;
	bFlagParaStructCopyWorking : BOOL; (*true, if cyclic para copying is active, 1 false cycle at every copy *)
	bStoreInitParaInDataObj : BOOL := FALSE;
	bTestflag : BOOL;
	bReadOutMETA_Once : BOOL;
	tParaCheck_iPvAdress : ARRAY[0..5] OF UDINT;
	tParaCheck_iPvLengt : ARRAY[0..5] OF UDINT;
	tParaCheck_rPvValue : ARRAY[0..5] OF REAL;
	tParaCheck_rRangeMIN : ARRAY[0..5] OF REAL;
	tParaCheck_rRangeMAX : ARRAY[0..5] OF REAL;
	tParaCheck_szPvName : ARRAY[0..5] OF STRING[35];
	ssFormatDetected : INT;
	szMetaDataPart : STRING[150];
	szFullTaskName : STRING[35];
	szFullMetaModuleName : STRING[35];
	debugLen : INT;
	debugSize : INT := 0;
	strcat_adr1 : UDINT;
	strcat_adr2 : UDINT;
	ssIndexTN : INT;
	bAlternate : BOOL;
	n : INT;
	iAlternateChecksum : DINT;
	iAlternateChecksumOld : DINT;
	ulDebugChkValue : ARRAY[0..999] OF UDINT;
	Adr1 : UDINT;
	Adr2 : UDINT;
	usPMWriteCntStepsize : UINT := 1; (*different step sizes to help debug*)
	usPMWriteCntXOR : UINT;
	usPMWriteCntAltSum : UINT;
	ulAdrPM : UDINT;
	usChkValuePM : USINT;
	ulAdrPara : UDINT;
	ulPara_len : UDINT;
	usChkValuePara : USINT;
	iDebugCountPMDifferences : DINT := 0;
	bEngineRunDetected : BOOL; (*detection status bit autocommand 100 /101  for engine run state*)
	ucMetaDataDebugInfoLine : ARRAY[0..24] OF STRING[80];
	ssIndexMand : INT := 0;
	szMetaDataMand : STRING[35];
	iMyErrorInfo_Autoreset : DINT; (*internal autoreset counter*)
	ssIndex_Version : INT; (*internal*)
	ssIndex_BU : INT; (*internal*)
	ssIndex_BU2 : INT; (*internal*)
END_VAR
```

### Program Logical/AuxiliariesGeneral/Pr_EO (IEC, version 4.13.0) - pressure engine oil

#### Pr_EO.st
```iecst
(*******************************************************************************
Pr_EO

This code is confidential and proprietary to the INNIO Company.
It may not be used in any form, or reproduced in any manner,
without the express written permission of the INNIO Company.
Copyright, INNIO Company, 2024

Customized modifications: -
------------------------

History:
-------
V3.90.0	20-03-2012	pankajrodey Created initial structured text code from ladder diagram
V3.99   28.02.2013	pankajrodey	Generated for modular software with changes for V3.30
		05.04.2013	lettenb.	oil filter pressure difference maximum alarm --> msg..
		28.05.2013	lettenb.	bTestEnabled Para -> loc.var
V4.04.0	25.10.2016	lettenb.	measuring signal plausibility check (Functional Safety EN 13849)
		07.08.2017	502423184	engine oil pressure after oil filter lowlow added FOR SWAT #3
V4.05.0	22.12.2017	lettenb.	comment added: Safety-related application software source code (EN 13849-1 / 4.6.3)
V4.07.0	25.04.2018	lettenb.	measuring signal plausibility check Pr_EOF_After(Functional Safety EN 13849)//SWAT920/5a
		13.06.2018	lettenb.	xTON_OilPressure added(acc.XT3), bugfix
                                xTON_ODR_AF_A: xTON_OilPressure.Q removed(only relevant for Pr_EngLubOil), bugfix
V4.09.0	22.04.2020	Schmid		corrected activation Z_ODR of A1017 oil pressure minimum due to change in tEng_Run.Do, bugfix
V4.13.0	05.03.2024	Tinello		Oil filter diff pressure monitoring (2023-184) - including issue #1122 and Fracas #3216

Instructions for use:
--------------------

Outstandings:
------------
(*******************************************************************************)

PROGRAM _CYCLIC

	(* delayed oil pressure signal failure *)
	xTON_OilPressure(IN:= NOT IN_AG.tPr_EngLubOil.GoodQual, PT:= T#0.3s);

	(* engine speed depending oil pressure limits *)
	xGR_MAXR_M_D800(In := IN_AG.rN_EngAct, Gw:= 800.0, Hy := 10.0);
	xTON_ODR_N(IN:= xGR_MAXR_M_D800.Q, PT:= T#10s);

	xSigScal_PrEO(X:= IN_AG.rN_EngAct, X1:= Para.rN_EOP_Lim1, Y1:= Para.rPr_EOP_LimSpeed1, X2:= Para.rN_EOP_Lim2, Y2:= Para.rPr_EOP_LimSpeed2);
	OUT_AG.rPr_EO_CalcLim := xSigScal_PrEO.Y_SCAL;

	IF xTON_ODR_N.Q THEN	OUT_AG.rPr_EO_Min := OUT_AG.rPr_EO_CalcLim;
	ELSE					OUT_AG.rPr_EO_Min := Para.rPr_EOP_LimSpeed1;
	END_IF;

	(********************************************************************************************************************
	Safety-related application software source code (EN 13849-1 / 4.6.3): BEGIN
	*********************************************************************************************************************)
	(* engine oil pressure lowlow *)
	xGR_MINR_ODRA(In:= IN_AG.tPr_EngLubOil.Ai, Gw:= OUT_AG.rPr_EO_Min, Hy:= Para.rPr_EOP_HyMin);
	xTON_ODRA(IN:= xGR_MINR_ODRA.Q AND IN_AG.tPB2MM.bParaSetupOk AND NOT xTON_OilPressure.Q, PT:= T#0.5s);
	AN_ODRA := xTON_ODRA.Q;

	(* engine oil pressure after oil filter lowlow *) (* SWAT #3 *)
	xGR_MINR_OD_AF_RA(In:= IN_AG.tPr_EOF_After.Ai, Gw:= OUT_AG.rPr_EO_Min, Hy:= Para.rPr_EOP_HyMin);
	xTON_ODR_AF_A(IN:= xGR_MINR_OD_AF_RA.Q AND IN_AG.tPB2MM.bParaSetupOk, PT:= T#0.5s);
	AN_OD_AF_RA := xTON_ODR_AF_A.Q;
	(********************************************************************************************************************
	Safety-related application software source code (EN 13849-1 / 4.6.3): END
	*********************************************************************************************************************)

	(* engine oil pressure low (warning) *)
	xGR_MINR_ODRW(In:= IN_AG.tPr_EngLubOil.Ai, Gw:= Para.rPr_EOP_LimSpeed2 + 0.2, Hy:= Para.rPr_EOP_HyMin);
	xTON_ODRW(IN:= xGR_MINR_ODRW.Q AND IN_AG.tPB2MM.bParaSetupOk AND NOT xTON_OilPressure.Q, PT:= T#0.5s);
	AN_ODRW := xTON_ODRW.Q;

	(* prelube pressure 1 (pump) *)
	xGR_MAXR_VSD1(In:= IN_AG.tPr_EngLubOil.Ai, Gw:= Para.rPr_Prel1EOP_LimHi, Hy:= Para.rPr_Prel1EOP_HyHi);
	xTON_VSD1(IN:= xGR_MAXR_VSD1.Q AND IN_AG.tPB2MM.bParaSetupOk, PT:= T#2s);
	OUT_AG.bPr_EOP_Prelub1 := xTON_VSD1.Q;

	(* prelube pressure 2 (pump) *)
	xGR_MAXR_VSD2(In:= IN_AG.tPr_EngLubOil.Ai, Gw:= Para.rPr_Prel2EOP_LimHi, Hy:= Para.rPr_Prel2EOP_HyHi);
	xTON_VSD2(IN:= xGR_MAXR_VSD2.Q AND IN_AG.tPB2MM.bParaSetupOk, PT:= T#2s);
	OUT_AG.bPr_EOP_Prelub2 	:= xTON_VSD2.Q;

	(* engine oil pressure limit 1 *)
	xGR_MAXR_PrEO_Hi1(In:= IN_AG.tPr_EngLubOil.Ai, Gw:= Para.rPr_EOP_Lim1, Hy:= Para.rPr_EOP_HyLim1);
	xTON_PrEO_Hi1(IN:= xGR_MAXR_PrEO_Hi1.Q AND IN_AG.tPB2MM.bParaSetupOk, PT:= T#2s);
	AN_ODGW1 :=   xTON_PrEO_Hi1.Q;

	(* engine oil pressure high *)
	xGR_MAXR_PrEO_Hi(In:= IN_AG.tPr_EngLubOil.Ai, Gw:= Para.rPr_EOP_LimMax, Hy:= Para.rPr_EOP_HyMax);
	xTON_PrEO_Hi(IN:= xGR_MAXR_PrEO_Hi.Q AND IN_AG.tPB2MM.bParaSetupOk AND NOT xTON_OilPressure.Q, PT:= T#30s);
	AN_ODR_MAX := xTON_PrEO_Hi.Q;

	(* engine oil pressure switch *)
	xGR_MAXR_DR_ODR(In:= IN_AG.rN_EngAct, Gw:= Para.rN_EOP_Lim1, Hy:= 10);
	OUT_AG.bPr_EOP_MonActive := xGR_MAXR_DR_ODR.Q AND IN_AG.tPB2MM.bParaSetupOk;

	(********************************************************************************************************************
	Safety-related application software source code (EN 13849-1 / 4.6.3): BEGIN
	*********************************************************************************************************************)
	(* engine oil pressure low - monitoring *)
	xTON_Z_ODR(IN:= OUT_AG.bPr_EOP_MonActive, PT:= T#3s);
	Z_ODR := xTON_Z_ODR.Q OR (IN_AG.tEng_Run.Do AND NOT IN_AG.bEng_MonOff);

	(* engine oil pressure low *)
	xGR_MAXR_ODR(In:= IN_AG.tPr_EngLubOil.Ai, Gw:= Para.rPr_EOP_LimSpeed2, Hy := 0);
	xTON_ODR(IN:= xGR_MAXR_ODR.Q, PT:= T#5s);
	xGR_MINR_DREHZ(In:= IN_AG.rN_EngAct, Gw := (Para.rN_EngNom - 100.0), Hy:= 0);

	xRS_FG_ODRUW(SET:= xTON_ODR.Q, RESET1:= xGR_MINR_DREHZ.Q);
	FG_ODRUW := xRS_FG_ODRUW.Q1;
	(********************************************************************************************************************
	Safety-related application software source code (EN 13849-1 / 4.6.3): END
	*********************************************************************************************************************)

	(* engine oil pressure high monitoring ON *)
	IF bTestEnabled THEN xTON_UW_ODR_MAX.PT:= T#1s;
	ELSE				 xTON_UW_ODR_MAX.PT:= T#600s;
	END_IF;
	xTON_UW_ODR_MAX(IN:= (xEngType.Type9 OR xEngType.Type6 OR xEngType.Type4 OR Para.bEngTyp3_Prelub_Active) AND M_DREHZ);
	UW_ODR_MAX := xTON_UW_ODR_MAX.Q;

	(*---------------------------------------------------------------------------*)
	(* measuring signal plausibility check - engine oil pressure (Functional Safety EN 13849) *)
	xTON_EngStop(IN:= 	NOT IN_AG.tEng_Run.Do
					AND NOT IN_AG.bEng_Aux_Dem_CDR
					AND NOT OUT_AG.tEOP1DC_Dem.Do
					AND NOT OUT_AG.tEOP1AC_Dem.Do
					AND NOT OUT_AG.tTC_EOP_On.Do, PT:= T#60s);
	xTON_EngRun(IN:= IN_AG.tEng_Run.Do, PT:= T#60s);

	xR_TRIG_StoreStopValue(CLK:= IN_AG.tPB2MM.bSys_Run AND xTON_EngStop.Q);
	xR_TRIG_StoreRunValue (CLK:= IN_AG.tPB2MM.bSys_Run AND xTON_EngRun.Q);

	IF xR_TRIG_StoreStopValue.Q THEN rPr_EO_StopValue := IN_AG.tPr_EngLubOil.Ai;
	END_IF;
	IF xR_TRIG_StoreRunValue.Q  THEN rPr_EO_RunValue  := IN_AG.tPr_EngLubOil.Ai;
	END_IF;
	IF bPr_EO_PcheckFail AND IN_AG.tAB2AG.bResetWarning THEN rPr_EO_StopValue := 0.0; (* reset *)
									                         rPr_EO_RunValue  := 0.0;
	END_IF;

	IF MM2VIS.bMsg2103             THEN				        bPr_EO_PcheckFail := FALSE;
	ELSIF (rPr_EO_StopValue = 0.0) THEN						bPr_EO_PcheckFail := FALSE; (* value not valid *)
	ELSIF (rPr_EO_RunValue  = 0.0) THEN						bPr_EO_PcheckFail := FALSE; (* value not valid *)
	ELSIF (rPr_EO_RunValue <= rPr_EO_StopValue) THEN		bPr_EO_PcheckFail := TRUE;
	ELSE
		IF (rPr_EO_RunValue - rPr_EO_StopValue) < 2.0 THEN	bPr_EO_PcheckFail := TRUE;
		END_IF;
	END_IF;

	(* measuring signal plausibility check - engine oil pressure after filter (Functional Safety EN 13849) *)//SWAT920/5a begin
	IF xR_TRIG_StoreStopValue.Q THEN rPr_EOaF_StopValue := IN_AG.tPr_EOF_After.Ai;
	END_IF;
	IF xR_TRIG_StoreRunValue.Q  THEN rPr_EOaF_RunValue  := IN_AG.tPr_EOF_After.Ai;
	END_IF;
	IF bPr_EOaF_PcheckFail AND IN_AG.tAB2AG.bResetWarning THEN rPr_EOaF_StopValue := 0.0; (* reset *)
									                           rPr_EOaF_RunValue  := 0.0;
	END_IF;

	IF MM2VIS.bMsg2432               THEN				        bPr_EOaF_PcheckFail := FALSE;
	ELSIF (rPr_EOaF_StopValue = 0.0) THEN						bPr_EOaF_PcheckFail := FALSE; (* value not valid *)
	ELSIF (rPr_EOaF_RunValue  = 0.0) THEN						bPr_EOaF_PcheckFail := FALSE; (* value not valid *)
	ELSIF (rPr_EOaF_RunValue <= rPr_EOaF_StopValue) THEN		bPr_EOaF_PcheckFail := TRUE;
	ELSE
		IF (rPr_EOaF_RunValue - rPr_EOaF_StopValue) < 2.0 THEN	bPr_EOaF_PcheckFail := TRUE;
		END_IF;
	END_IF; 	//SWAT920/5a end

	(*--------------------------------------------------*)
	(* Measurement monitoring - oil pressure 			*)
	(*--------------------------------------------------*)
	bAMM_Pr_bEOF_Ms			:= Para.b_EOF_DiffMonActive		AND NOT IN_AG.tPr_EOF_DiffMon.GoodQual;							(* A2242 *)
	bAMM_Pr_aEOF_Ms			:= Para.bPr_EOF_After_Active	AND NOT IN_AG.tPr_EOF_After.GoodQual;							(* A2260 *)(* W2432 *)
	bAMM_Pr_EngLubOil_Ms	:= 									NOT IN_AG.tPr_EngLubOil.GoodQual;							(* A2260 *)

		bRelMon_Pr_bEOF		:= Para.b_EOF_DiffMonActive  	AND NOT bAMM_Pr_bEOF_Ms;
		bRelMon_Pr_aEOF		:= Para.bPr_EOF_After_Active  	AND NOT bAMM_Pr_aEOF_Ms;
		bRelMon_Pr_EngLubOil:= 									NOT bAMM_Pr_EngLubOil_Ms;

	(*--------------------------------------------------*)
	(* Oil filter differential pressure					*)
	(*--------------------------------------------------*)
	IF 	  NOT bRelMon_Pr_bEOF 		THEN rDPr_EOF	:= 0;													(* NO signal before filter available *)
	ELSE
		IF 	  bRelMon_Pr_aEOF 		THEN rDPr_EOF	:= IN_AG.tPr_EOF_DiffMon.Ai - IN_AG.tPr_EOF_After.Ai;	(* before filter - after filter *)
		ELSIF bRelMon_Pr_EngLubOil	THEN rDPr_EOF	:= IN_AG.tPr_EOF_DiffMon.Ai - IN_AG.tPr_EngLubOil.Ai; 	(* before filter - last lubr. point *)
									ELSE rDPr_EOF	:= 0;													(* NO signal after filter available *)
		END_IF
	END_IF

	xGR_MAXR_DPr_EOF_Limit1(In:= rDPr_EOF, Gw:= MAX(0.11, Para.rPr_EOF_DiffMonLimit1), Hy:= 0.1); 	(* 0.11 to avoid error because of wrong para setting *)
	xGR_MAXR_DPr_EOF_Limit2(In:= rDPr_EOF, Gw:= MAX(0.11, Para.rPr_EOF_DiffMonLimit2), Hy:= 0.1); 	(* Hysteresis 0.1 bar *)
	xGR_MAXR_DPr_EOF_Limit3(In:= rDPr_EOF, Gw:= MAX(0.11, Para.rPr_EOF_DiffMonLimit3), Hy:= 0.1);

	bAMM_DPr_EOF_Lim1	:= (IN_AG.tT_EO.Ai > Para.rT_EOF_DiffMonRel) AND NOT MM2VIS.bMsg2102 AND xGR_MAXR_DPr_EOF_Limit1.Q;	(* W3414 *)
	bAMM_DPr_EOF_Lim2	:= (IN_AG.tT_EO.Ai > Para.rT_EOF_DiffMonRel) AND NOT MM2VIS.bMsg2102 AND xGR_MAXR_DPr_EOF_Limit2.Q;	(* W3415 *)
	bAMM_DPr_EOF_Lim3	:= (IN_AG.tT_EO.Ai > Para.rT_EOF_DiffMonRel) AND NOT MM2VIS.bMsg2102 AND xGR_MAXR_DPr_EOF_Limit3.Q;	(* A1059 *)
END_PROGRAM
```

#### Pr_EO.var
```iecst
VAR
	xGR_MAXR_VSD2 : GR_MAXR;
	xGR_MAXR_M_D800 : GR_MAXR;
	xGR_MAXR_VSD1 : GR_MAXR;
	xGR_MAXR_PrEO_Hi1 : GR_MAXR;
	xGR_MAXR_PrEO_Hi : GR_MAXR;
	xGR_MAXR_ODR : GR_MAXR;
	xGR_MAXR_DR_ODR : GR_MAXR;
	xGR_MINR_ODRW : GR_MINR;
	xGR_MINR_ODRA : GR_MINR;
	xGR_MINR_DREHZ : GR_MINR;
	xRS_FG_ODRUW : RS;
	xTON_VSD2 : TON;
	xTON_PrEO_Hi1 : TON;
	xTON_Z_ODR : TON;
	xTON_VSD1 : TON;
	xTON_UW_ODR_MAX : TON;
	xTON_PrEO_Hi : TON;
	xTON_OilPressure : TON;
	xTON_ODR : TON;
	xTON_ODRW : TON;
	xTON_ODR_N : TON;
	xTON_ODRA : TON;
	xSigScal_PrEO : xSigScal_R;
	rPr_EO_StopValue : REAL := 0.0;
	xR_TRIG_StoreStopValue : R_TRIG;
	rPr_EO_RunValue : REAL := 0.0;
	xR_TRIG_StoreRunValue : R_TRIG;
	xTON_EngStop : TON;
	xTON_EngRun : TON;
	xGR_MINR_OD_AF_RA : GR_MINR;
	xTON_ODR_AF_A : TON;
	rPr_EOaF_StopValue : REAL := 0.0; (*SWAT920/5*)
	rPr_EOaF_RunValue : REAL := 0.0; (*SWAT920/5*)
	xGR_MAXR_DPr_EOF_Limit1 : GR_MAXR; (*FuB*)
	xGR_MAXR_DPr_EOF_Limit2 : GR_MAXR; (*FuB*)
	xGR_MAXR_DPr_EOF_Limit3 : GR_MAXR; (*FuB*)
	bRelMon_Pr_bEOF : BOOL; (*Release monitoring - oil pressure before oil filter*)
	bRelMon_Pr_aEOF : BOOL; (*Release monitoring - oil pressure after oil filter*)
	bRelMon_Pr_EngLubOil : BOOL; (*Release monitoring - oil pressure engine lube oil*)
END_VAR
```

### Program Logical/AuxiliariesGeneral/T_EO_AG (IEC, version 4.06.0) - temperature engine oil

#### T_EO_AGCyclic.st
```iecst
(*******************************************************************************
T_EO	engine oil temperature

This code is confidential and proprietary to the INNIO Company.
It may not be used in any form, or reproduced in any manner, without the express
written permission of the INNIO Company.
Copyright, INNIO Company, 2019

Customized modifications:
-------------------------
-

History:
--------
V0.1	02.10.1998	Pa			erstellt
		26.11.1998	Pa			korrekturlesung
V1.70	04.04.2002	LH			Verzögerung Öltemperatur max. => 5min
								Grenzwert Öltemperatur max. + 4/5°C (Abstellung)
V1.80	06.02.2003	LH			Grenzwert Öltemperatur max. + 4°C --> + 2°C (BR 2/3/4)
		06.03.2003	LH			VISU-Grenzwerte erst aktiv wenn Rezepte auf Steuerung sind
		18.03.2003	LH			Einlesen Analogeingang --> pb17
V3.20.0	12.05.2010	lettenb.	OT_LFG added for BR9
		01.07.2010 				Öltemperatur maximum: BR9_B added
V3.90.0	06.12.2011	Ganguly		generated from otpCyclic.st V3.20
		08.03.2012	Denk		review and clean-up
V3.99.0	04.04.2013	lettenb.	INIT removed (no write to parameter allowed)
		28.05.2013	lettenb.	bTestEnabled Para -> loc.var
		29.07.2013				engine oil temp.high monitoring moved to MsgAG
V4.06.0	29.08.2018	Perktold	added fast start release from oil temperature

Instructions for use:
--------------------
Outstandings:
------------
********************************************************************)

PROGRAM _CYCLIC

	(* load release from oil temperature *)
	xGR_MAXR_OT_LFG(In:= IN_AG.tT_EO.Ai, Gw:= Para.rT_EOP_LimRelLoad, Hy:= Para.rT_EOP_HyRelLoad);
	xTON_OT_LFG(IN:= IN_AG.tPB2MM.bParaSetupOk AND xGR_MAXR_OT_LFG.Q, PT:= T#2s);
	OUT_AG.bT_EOP_RelLoad := xTON_OT_LFG.Q;

	(* fast start release from oil temperature *)
	xGR_MAXR_OT_FS(In:= IN_AG.tT_EO.Ai, Gw:= 27.0, Hy:= 1.0);
	xTON_OT_FS(IN:= IN_AG.tPB2MM.bParaSetupOk AND xGR_MAXR_OT_FS.Q, PT:= T#2s);
	OUT_AG.bT_EOP_RelFS := xTON_OT_FS.Q;

	(*-------------------------------------------------------------------------------*)
	(* power reduction according high oil temperature *)
	OUT_AG.rP_Red_T_Oil_Norm := LIMIT(0.5, (1 - ((IN_AG.tT_EO.Ai - Para.rP_Red_T_Oil_Start) * Para.rP_Red_T_Oil_Rate)), 1.0);

END_PROGRAM
```

#### T_EO_AG.var
```iecst
VAR
	xGR_MAXR_OT_LFG : GR_MAXR;
	xTON_OT_LFG : TON;
	xGR_MAXR_OT_FS : GR_MAXR;
	xTON_OT_FS : TON;
END_VAR
```

### Program Logical/AuxiliariesGeneral/TrP_red (IEC, version 4.04.0) - transformer power reduction
